// SIMATIC S7-200 project (STEP 7-Micro/WIN), CPU 226 CN REL 02.01

SYMBOL_TABLE 用户定义1
T_177            T177     // M25.1动作计时(2)
T_59             T59      // Y轴原点行程开关动作计时
T_83             T83      // M25.1动作计时(1)
T_71             T71      // M28.1动作计时(3)
T_70             T70      // M28.1动作计时(2)
T_69             T69      // M28.1动作计时(1)
T_185            T185     // PH1动作计时
T_180            T180     // PH2不动作计时
T_190            T190     // SL5动作延时
T_81             T81      // M26.0动作计时
T_82             T82      // 夹紧装置电磁阀松开线圈动作计时
SA2              I0.0     // 1=板链线与机械手联锁,0=板链线单独
SF3              I0.1     // 板链线/机械手联锁启动
SS3              I0.2     // 板链线/机械手联锁停止
SB_1             I0.3     // 板链线反转点动
SB_2             I0.4     // X轴Y轴伺服回原点
SB_3             I0.5     // 故障解除
KA1              I0.6     // 板链线变频故障
PH1              I0.7     // 板链线产品到位
PH2              I1.0     // 差速链工装板有无产品
SL1              I1.1     // X轴伺服左极限
SL2              I1.2     // X轴伺服原点(常闭触点输入)
SL3              I1.3     // X轴伺服右极限
SL4              I1.4     // Y轴伺服上极限
SL5              I1.5     // Y轴伺服原点(常闭触点输入)
SL6              I1.6     // Y轴伺服下极限
SL7              I1.7     // 板链线夹具到位
SL8              I2.0     // 板链线下线保护
SL11             I2.1     // 差速链线工装板后边沿
SL12             I2.2     // 差速链线工装板前边沿
SP1              I2.3     // Y轴提升气缸提升到位
SP2              I2.4     // Y轴提升气缸下降到位
SP3              I2.5     // Y轴旋转气缸旋转到位
SP4              I2.6     // Y轴旋转气缸复位到位
SP5              I2.7     // X轴旋转气缸旋转到位
ASD1_SRDY        I3.0     // X轴伺服准备完毕
ASD1_ZSPD        I3.1     // X轴伺服零速状态
ASD1_TPOS        I3.2     // X轴伺服位置软限位
ASD1_ALRM        I3.3     // X轴伺服报警
ASD2_SRDY        I3.4     // Y轴伺服准备完毕
ASD2_ZSPD        I3.5     // Y轴伺服零速状态
ASD2_TPOS        I3.6     // Y轴伺服位置软限位
ASD2_ALRM        I3.7     // Y轴伺服报警
SP6              I4.0     // X轴旋转气缸复位到位
SP7              I4.1     // 抓紧气缸抓紧(1)
SP8              I4.2     // 抓紧气缸抓紧(2)
SP9              I4.3     // 抓紧气缸抓紧(3)
SP10             I4.4     // 抓紧气缸抓紧(4)
SP11_14          I4.5     // 抓紧气缸松开
KP1              I4.6     // 压力过低报警
SJ1_7            I4.7     // 板链线/机械手急停
M0_0             M0.0     // 板链线/机械手联锁投入
M0_2             M0.2     // 板链线/机械手联锁运行上升延微分
M0_3             M0.3     // 板链线单独正转投入
M0_6             M0.6     // 故障蜂鸣告警
M0_7             M0.7     // 紧急停止蜂鸣告警
M1_0             M1.0     // 气压过低蜂鸣报警
M1_1             M1.1     // 蜂鸣报警消音
M1_2             M1.2     // 故障/气压过低蜂鸣报警汇总
M3_7             M3.7     // Y轴伺服在板链线/差速链线上空下移脉冲数逻辑运算错误
M4_0             M4.0     // 机械手Y轴伺服空闲位下降沿微分
M4_1             M4.1     // Y轴伺服在板链线上空下移动作保持
M5_1             M5.1     // Q0.0脉冲输出指令
M5_2             M5.2     // Q0.1脉冲输出指令
M7_1             M7.1     // M14.1下降沿微分
M7_2             M7.2     // 机械手总复位结束信号
M9_1             M9.1     // Q0.0脉冲控制子程序PTO0_CTRL的I_STOP参数
M9_2             M9.2     // Q0.0脉冲控制子程序PTO0_CTRL的D_STOP参数
M10_0            M10.0    // Q0.0脉冲控制子程序PTO0_CTRL执行完成标志
M11_0            M11.0    // 机械手点动模式
M11_3            M11.3    // X轴伺服点动
M11_4            M11.4    // Y轴伺服点动
M12_0            M12.0    // XY轴伺服原点回归点动
M12_1            M12.1    // X轴伺服原点回归点动
M12_2            M12.2    // Y轴伺服原点回归点动
M12_3            M12.3    // XY轴伺服原点回归停止
M12_4            M12.4    // X轴伺服原点回归保持
M12_5            M12.5    // Y轴伺服原点回归保持
M12_6            M12.6    // 机械手总复位
M12_7            M12.7    // 机械手总复位停止
M13_0            M13.0    // 机械手总复位进行中
M13_1            M13.1    // X轴伺服运行指示
M13_2            M13.2    // Y轴伺服运行指示
M14_0            M14.0    // Y轴提升气缸提升
M14_1            M14.1    // Y轴提升气缸下降
M14_2            M14.2    // Y轴旋转气缸旋转
M14_3            M14.3    // Y轴旋转气缸复位
M14_4            M14.4    // X轴旋转气缸旋转
M14_5            M14.5    // X轴旋转气缸复位
M14_6            M14.6    // 抓取气缸抓紧
M14_7            M14.7    // 抓取气缸松开
M15_0            M15.0    // X轴伺服回原点
M15_1            M15.1    // Y轴伺服回原点
M16_0            M16.0    // X轴从板链线上空移向差速链上空状态保持
M16_1            M16.1    // X轴走到一定位置时Y轴旋转没有到位则停止X轴移向差速链
M16_2            M16.2    // X轴走到一定位置时X轴旋转没有到位则停止X轴移向差速链
M16_3            M16.3    // X轴没有走到一定位置时不允许提升气缸下降
M17_0            M17.0    // 板链线/机械手联锁投入
M17_1            M17.1    // 联锁运行状态
M17_2            M17.2    // 板链线运行状态指示
M17_3            M17.3    // 设备故障指示
M17_4            M17.4    // 触摸屏紧急停止
M17_5            M17.5    // 控制柜硬急停/触摸屏软急停汇总
M17_6            M17.6    // 触摸屏上设备启动
M17_7            M17.7    // 触摸屏上设备停止
M18_0            M18.0    // 触摸屏上板链线反转点动
M18_1            M18.1    // 触摸屏上故障解除
M18_2            M18.2    // 触摸屏上报警消音
M18_3            M18.3    // 机械手X轴伺服空闲位(0=PTO忙,1=PTO空闲)
M18_4            M18.4    // 机械手Y轴伺服空闲位(0=PTO忙,1=PTO空闲)
M18_5            M18.5    // 触摸屏上机械手X轴伺服方向(0=移向差速链线,1=移向板链线)
M18_6            M18.6    // 触摸屏上机械手Y轴伺服方向(0=下移,1=上移)
M19_1            M19.1    // Q0.1脉冲控制子程序PTO1_CTRL的I_STOP参数
M19_2            M19.2    // Q0.1脉冲控制子程序PTO1_CTRL的D_STOP参数
M20_0            M20.0    // Q0.1脉冲控制子程序PTO1_CTRL执行完成标志
M21_0            M21.0    // 板链线夹具前边沿到位
M21_1            M21.1    // 机械手抓紧气缸抓紧
M21_2            M21.2    // 联锁运行时Y轴提升气缸提升保持
M22_1            M22.1    // 抓紧气缸抓紧磁性开关(1)已经动作
M22_2            M22.2    // 抓紧气缸抓紧磁性开关(2)已经动作
M22_3            M22.3    // 抓紧气缸抓紧磁性开关(3)已经动作
M22_4            M22.4    // 抓紧气缸抓紧磁性开关(4)已经动作
M22_5            M22.5    // 抓紧气缸4个抓紧检测磁性开关已经动作
M22_6            M22.6    // 抓紧气缸4个抓紧检测磁性开关已经动作上升延
M22_7            M22.7    // Y轴提升气缸缩回保持
M23_0            M23.0    // 板链线停车等待差速链空工装板到位
M23_1            M23.1    // X轴伺服右移/X轴旋转气缸旋转/Y轴旋转气缸旋转
M24_0            M24.0    // X轴伺服右移到位
M24_1            M24.1    // Y轴伺服电机下移(3种产品3种位置,大约20mm左右)
M24_2            M24.2    // Y轴伺服在差速链上空从当前位置移至对应产品处
M24_3            M24.3    // Y轴伺服空闲上升延微分
M24_7            M24.7    // 点动模式上升沿微分
M25_0            M25.0    // Y轴伺服下移到位
M25_1            M25.1    // 夹紧装置电磁阀松开线圈动作保持
M26_0            M26.0    // Y轴伺服上移到原点
M26_1            M26.1    // 抓紧气缸松开上升延
M26_2            M26.2    // Y轴伺服下移方向信号
M27_0            M27.0    // Y轴伺服上移到位
M28_0            M28.0    // X轴伺服左移
M28_1            M28.1    // X轴原点回归信号保持
M28_3            M28.3    // Y轴原点回归信号保持
M29_0            M29.0    // Y轴伺服回原点后再下降到对应的Y轴高度
M30_0            M30.0    // 机械手处于初始状态
M31_0            M31.0    // 差速链阻挡器电磁阀下降线圈得电保持
M31_6            M31.6    // 手动停止PTO0脉冲输出标志
M31_7            M31.7    // 手动停止PTO0脉冲输出标志
ASD1_PLS         Q0.0     // X轴伺服位置脉冲
ASD2_PLS         Q0.1     // Y轴伺服位置脉冲
ASD1_SIGN        Q0.2     // X轴伺服方向(0=移向差速链线,1=移向板链线)
ASD2_SIGN        Q0.3     // Y轴伺服方向(0=下移,1=上移)
KA2              Q0.7     // 设备启动/故障蜂鸣告警
KA3              Q1.0     // 板链线运行状态
KA4              Q1.1     // 板链线变频器正转
KA5              Q1.2     // 板链线变频器反转
KA6              Q1.3     // 板链线/机械手联锁运行状态
KA7              Q1.4     // 机械手紧急停止
KA8              Q1.5     // Y轴提升气缸提升
KA9              Q1.6     // Y轴提升气缸下降
KA10             Q1.7     // 故障闪光告警
YV2_1            Q2.0     // Y轴旋转气缸旋转
YV2_2            Q2.1     // Y轴旋转气缸复位
YV3_1            Q2.2     // X轴旋转气缸旋转
YV3_2            Q2.3     // X轴旋转气缸复位
YV4_1            Q2.4     // 抓取气缸抓紧
YV4_2            Q2.5     // 抓取气缸松开
YV11             Q2.6     // 差速链线前阻挡器
YV12             Q2.7     // 差速链线后阻挡器
ASD1启动           Q3.0     // X轴伺服启动
ASD1脉冲清除         Q3.1     // X轴伺服脉冲清除
ASD1原点回归         Q3.2     // X轴伺服原点回归
ASD1故障复位         Q3.3     // X轴伺服故障复位
ASD2启动           Q3.4     // Y轴伺服启动
ASD2脉冲清除         Q3.5     // Y轴伺服脉冲清除
ASD2原点回归         Q3.6     // Y轴伺服原点回归
ASD2故障复位         Q3.7     // Y轴伺服故障复位
SM0_0            SM0.0    // 该位始终为1
SM0_1            SM0.1    // 第一个扫描周期为1
SM66_7           SM66.7   // PTO0空闲位：0=PTO忙，1=PTO空闲
SM67_7           SM67.7   // PTO0/PWM0有效位：1=有效
SM76_7           SM76.7   // PTO1空闲位：0=PTO忙，1=PTO空闲
SM77_7           SM77.7   // PTO1/PWM1有效位：1=有效
SMD_72           SMD72    // PTO0脉冲计数值
SMD_82           SMD82    // PTO1脉冲计数值
SMW_68           SMW68    // PTO0/PWM0周期
SMW_78           SMW78    // PTO1/PWM1周期
T_37             T37      // 板链线/机械手启动告警时间
T_38             T38      // 板链线单独正转启动告警时间
T_39             T39      // 故障蜂鸣报警之静音时间
T_40             T40      // 故障蜂鸣报警之鸣音时间
T_41             T41      // 急停蜂鸣报警之静音时间
T_42             T42      // 急停蜂鸣报警之鸣音时间
T_43             T43      // 气压过低蜂鸣报警之静音时间
T_44             T44      // 气压过低蜂鸣报警之鸣音时间
T_46             T46      // 下线保护光电开关动作计时
T_51             T51      // 夹紧电磁阀夹紧动作时间
T_54             T54      // X轴右移到位信号保持时间
T_55             T55      // 夹紧装置电磁阀松开线圈动作时间
T_57             T57      // X轴伺服左移延时
T_58             T58      // 原点行程开关动作时间
T_61             T61      // 差速链阻挡器电磁阀下降线圈得电时间
T_111            T111     // XY轴伺服加减速用的时钟脉冲
T_112            T112     // Y轴伺服点动计时
T_115            T115     // 触摸屏上板链线运行动画图片切换时间
T_131            T131     // YV4-1动作计时
T_132            T132     // Y轴提升气缸提升动作计时(1)
T_133            T133     // Y轴提升气缸提升动作计时(2)
T_134            T134     // YV3-1动作计时
T_135            T135     // M24.1动作计时
T_136            T136     // Y轴伺服上移计时
T_157            T157     // 机械手总复位时到达X轴Y轴原点计时
T_158            T158     // M4.1动作计时
T_175            T175     // 机械手到达Y轴原点计时
T_200            T200     // Y轴下移到位信号保持时间
T_210            T210     // 紧急停止复位后（就是解除了紧急停止）计时
T_247            T247     // 联锁运行计时
V308_1           V308.1   // Q0.0脉冲手动模式子程序PTO0_MAN的Run/Stop参数
V1308_1          V1308.1  // Q0.1脉冲手动模式子程序PTO1_MAN的Run/Stop参数
VB_1             VB1      // 变频器频率检测方式(VB1=0自动检测,VB1=1手动给定)
VB_300           VB300    // Q0.0脉冲控制子程序PTO0_CTRL的错误代码
VB_314           VB314    // Q0.0脉冲手动模式子程序PTO0_MAN的错误代码
VB_1300          VB1300   // Q0.1脉冲控制子程序PTO1_CTRL的错误代码
VB_1314          VB1314   // Q0.1脉冲手动模式子程序PTO1_MAN的错误代码
VD_108           VD108    // PLC自动检测到的变频器频率值
VD_150           VD150    // 手动给定的变频器的当前频率值
VD_154           VD154    // 变频器的有效当前频率值
VD_160           VD160    // 产品种类(1小号,2中号,3大号,4自定义)
VD_164           VD164    // 小号产品的中心高度
VD_168           VD168    // 小号产品的半径
VD_172           VD172    // 中号产品的中心高度
VD_176           VD176    // 中号产品的半径
VD_180           VD180    // 大号产品的中心高度
VD_184           VD184    // 大号产品的半径
VD_188           VD188    // 自定义产品的长度
VD_192           VD192    // 自定义产品的直径
VD_196           VD196    // 当前有效产品的长度
VD_200           VD200    // 当前有效产品的半径
VD_294           VD294    // PTO0脉冲计数值
VD_302           VD302    // Q0.0脉冲控制子程序PTO0_CTRL的C_Pos参数
VD_310           VD310    // Q0.0脉冲手动模式子程序PTO0_MAN的Speed参数
VD_316           VD316    // Q0.0脉冲手动模式子程序PTO0_MAN的C_Pos参数
VD_1294          VD1294   // PTO1脉冲计数值
VD_1302          VD1302   // Q0.1脉冲控制子程序PTO1_CTRL的C_Pos参数
VD_1310          VD1310   // Q0.1脉冲手动模式子程序PTO1_MAN的Speed参数
VD_1316          VD1316   // Q0.1脉冲手动模式子程序PTO1_MAN的C_Pos参数
VD_1900          VD1900   // 机械手X轴与板链线运行速度相等时X轴伺服脉冲与变频器频率的比值
VD_1904          VD1904   // 机械手X轴与板链线运行速度相等时X轴伺服脉冲的频率
VD_2000          VD2000   // 机械手X轴与板链线同步时的PTO0周期值(微秒，实数)
VD_2004          VD2004   // 机械手X轴与板链线同步时的PTO0周期计算中间值1
VD_2008          VD2008   // 机械手X轴与板链线同步时的PTO0周期计算中间值2
VD_2012          VD2012   // 机械手X轴与板链线同步时的PTO0周期值(微秒,双整数)
VD_3000          VD3000   // 机械手在X轴方向每行走1mm，需要给X轴伺服电机的脉冲数(实数)
VD_3004          VD3004   // 机械手X轴与板链线同步的行走需要的脉冲数(实数)
VD_3008          VD3008   // 机械手X轴与板链线同步的行走需要的脉冲数(双整数)
VD_3016          VD3016   // X轴伺服跟随板链线行走完成后到移动到位需要的脉冲数(实数)
VD_3020          VD3020   // X轴伺服跟随板链线行走完成后到移动到位需要的脉冲数(双整数)
VD_4000          VD4000   // 机械手在Y轴方向每行走1mm，需要给Y轴伺服电机的脉冲数
VD_5000          VD5000   // 小号产品对应的Y轴伺服电机脉冲数(实数)
VD_5004          VD5004   // 小号产品对应的Y轴伺服电机脉冲数(双整数)
VD_5008          VD5008   // 在差速链上空各种产品对应的机械手Y轴下移脉冲数
VD_5020          VD5020   // 中号产品对应的Y轴伺服电机脉冲数(实数)
VD_5024          VD5024   // 中号产品对应的Y轴伺服电机脉冲数(双整数)
VD_5040          VD5040   // 大号产品对应的Y轴伺服电机脉冲数(实数)
VD_5044          VD5044   // 大号产品对应的Y轴伺服电机脉冲数(双整数)
VD_5052          VD5052   // 在差速链线上空各种产品对应的机械手Y轴下移脉冲数(电子齿轮比分子为3)
VD_6004          VD6004   // 小号产品对应的在板链线上空的Y轴伺服脉冲数(实数)
VD_6008          VD6008   // 小号产品对应的在板链线上空的Y轴伺服脉冲数(双整数)
VD_6012          VD6012   // 在板链链线上空各种产品对应的机械手Y轴下移脉冲数(电子齿轮比分子为1)
VD_6016          VD6016   // 在板链链线上空各种产品对应的机械手Y轴下移脉冲数(电子齿轮比分子为3)
VD_6024          VD6024   // 中号产品对应的在板链线上空的Y轴伺服脉冲数(实数)
VD_6028          VD6028   // 中号产品对应的在板链线上空的Y轴伺服脉冲数(双整数)
VD_6044          VD6044   // 大号产品对应的在板链线上空的Y轴伺服脉冲数(实数)
VD_6048          VD6048   // 大号产品对应的在板链线上空的Y轴伺服脉冲数(双整数)
VW_290           VW290    // PTO0/PWM0周期
VW_1290          VW1290   // PTO1/PWM1周期
VW_2020          VW2020   // 机械手X轴与板链线同步时的PTO0周期值(微秒，整数)
VW_7080          VW7080   // 触摸屏上板链线运行动画状态存储器
VW_7090          VW7090   // 触摸屏上机械手运行动画状态存储器
END_SYMBOL_TABLE

ORGANIZATION_BLOCK 总体控制:OB1
TITLE=总体控制；
BEGIN
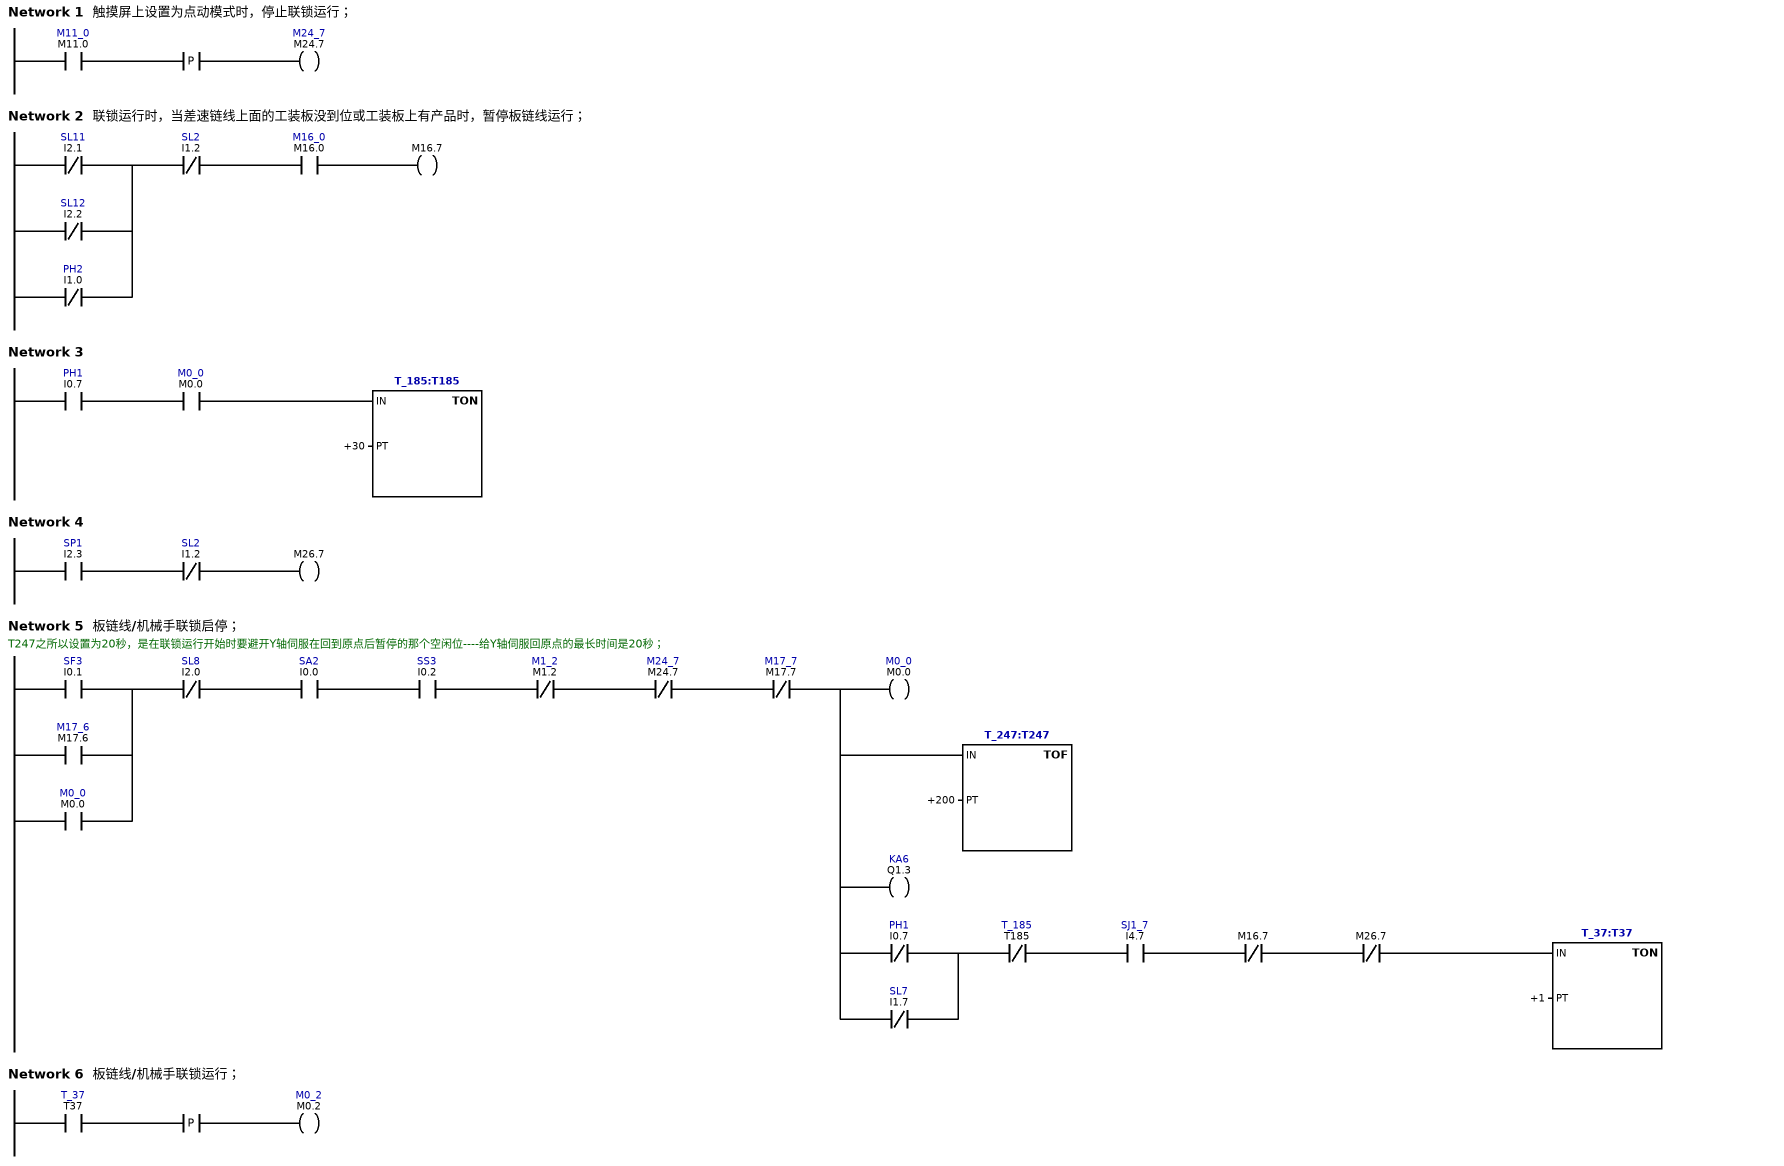
Network 1 // 触摸屏上设置为点动模式时，停止联锁运行；
LD     M11_0:M11.0
EU
=      M24_7:M24.7
Network 2 // 联锁运行时，当差速链线上面的工装板没到位或工装板上有产品时，暂停板链线运行；
LDN    SL11:I2.1
ON     SL12:I2.2
ON     PH2:I1.0
AN     SL2:I1.2
A      M16_0:M16.0
=      M16.7
Network 3
LD     PH1:I0.7
A      M0_0:M0.0
TON    T_185:T185, +30
Network 4
LD     SP1:I2.3
AN     SL2:I1.2
=      M26.7
Network 5 // 板链线/机械手联锁启停；
// T247之所以设置为20秒，是在联锁运行开始时要避开Y轴伺服在回到原点后暂停的那个空闲位----给Y轴伺服回原点的最长时间是20秒；
LD     SF3:I0.1
O      M17_6:M17.6
O      M0_0:M0.0
AN     SL8:I2.0
A      SA2:I0.0
A      SS3:I0.2
AN     M1_2:M1.2
AN     M24_7:M24.7
AN     M17_7:M17.7
=      M0_0:M0.0
TOF    T_247:T247, +200
=      KA6:Q1.3
LDN    PH1:I0.7
ON     SL7:I1.7
ALD
AN     T_185:T185
A      SJ1_7:I4.7
AN     M16.7
AN     M26.7
TON    T_37:T37, +1
Network 6 // 板链线/机械手联锁运行；
LD     T_37:T37
EU
=      M0_2:M0.2
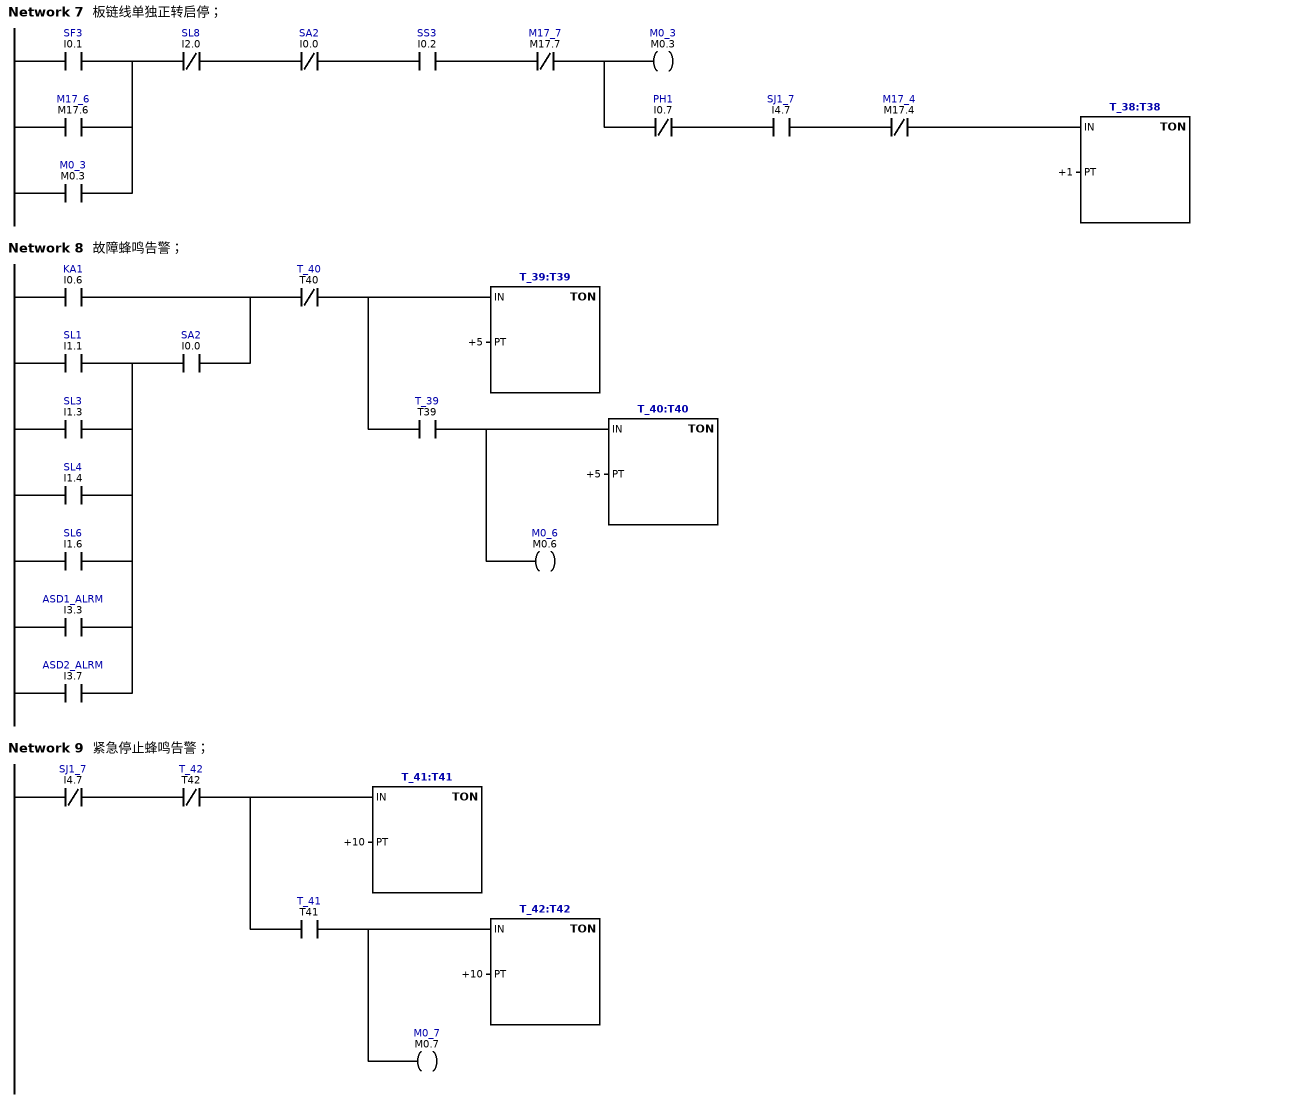
Network 7 // 板链线单独正转启停；
LD     SF3:I0.1
O      M17_6:M17.6
O      M0_3:M0.3
AN     SL8:I2.0
AN     SA2:I0.0
A      SS3:I0.2
AN     M17_7:M17.7
=      M0_3:M0.3
AN     PH1:I0.7
A      SJ1_7:I4.7
AN     M17_4:M17.4
TON    T_38:T38, +1
Network 8 // 故障蜂鸣告警；
LD     KA1:I0.6
LD     SL1:I1.1
O      SL3:I1.3
O      SL4:I1.4
O      SL6:I1.6
O      ASD1_ALRM:I3.3
O      ASD2_ALRM:I3.7
A      SA2:I0.0
OLD
AN     T_40:T40
TON    T_39:T39, +5
A      T_39:T39
TON    T_40:T40, +5
=      M0_6:M0.6
Network 9 // 紧急停止蜂鸣告警；
LDN    SJ1_7:I4.7
AN     T_42:T42
TON    T_41:T41, +10
A      T_41:T41
TON    T_42:T42, +10
=      M0_7:M0.7
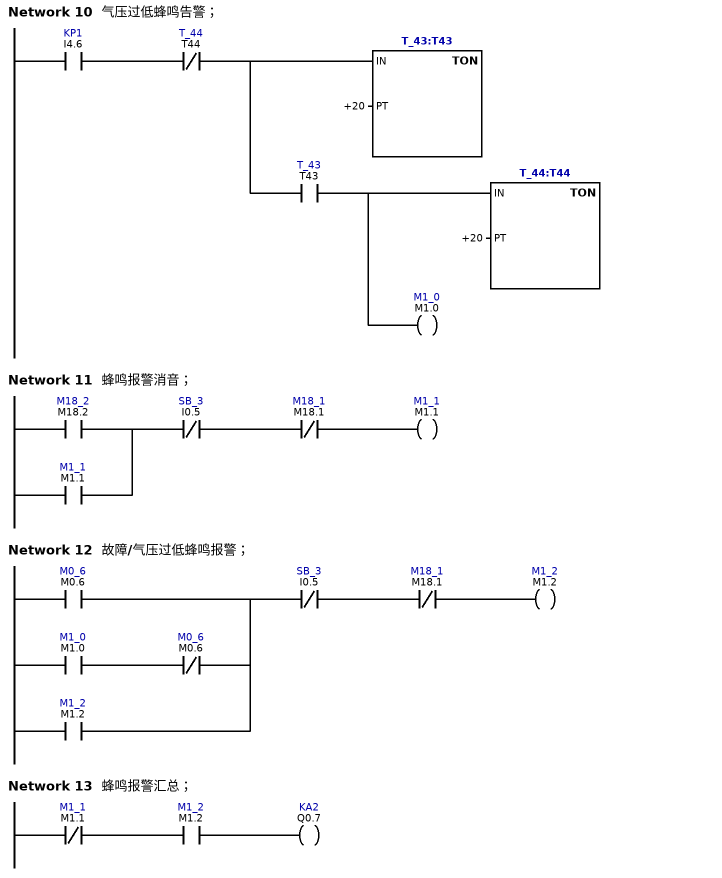
Network 10 // 气压过低蜂鸣告警；
LD     KP1:I4.6
AN     T_44:T44
TON    T_43:T43, +20
A      T_43:T43
TON    T_44:T44, +20
=      M1_0:M1.0
Network 11 // 蜂鸣报警消音；
LD     M18_2:M18.2
O      M1_1:M1.1
AN     SB_3:I0.5
AN     M18_1:M18.1
=      M1_1:M1.1
Network 12 // 故障/气压过低蜂鸣报警；
LD     M0_6:M0.6
LD     M1_0:M1.0
AN     M0_6:M0.6
OLD
O      M1_2:M1.2
AN     SB_3:I0.5
AN     M18_1:M18.1
=      M1_2:M1.2
Network 13 // 蜂鸣报警汇总；
LDN    M1_1:M1.1
A      M1_2:M1.2
=      KA2:Q0.7
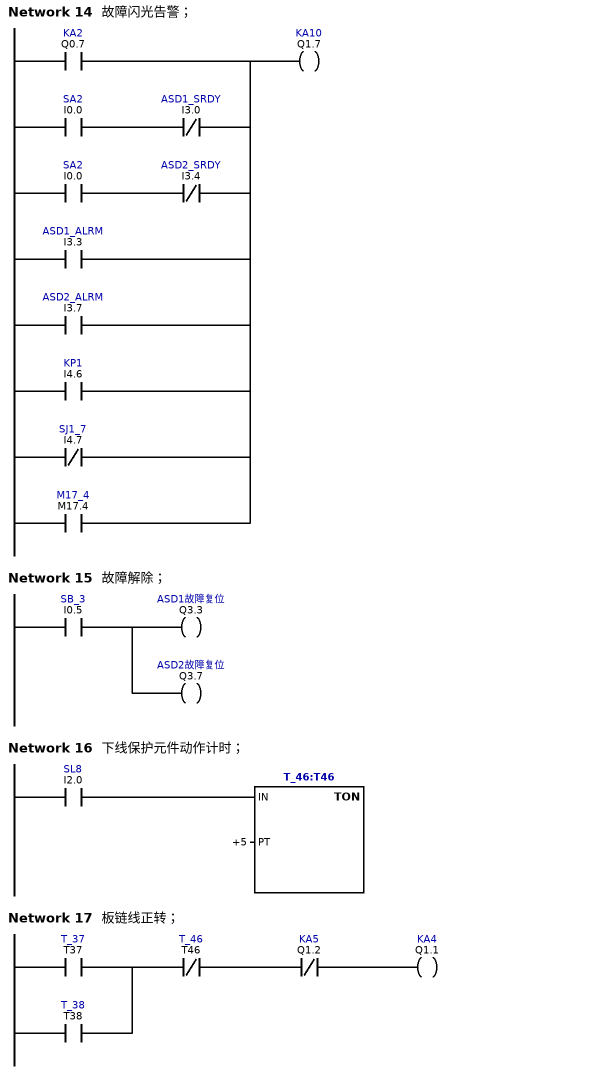
Network 14 // 故障闪光告警；
LD     KA2:Q0.7
LD     SA2:I0.0
AN     ASD1_SRDY:I3.0
OLD
LD     SA2:I0.0
AN     ASD2_SRDY:I3.4
OLD
O      ASD1_ALRM:I3.3
O      ASD2_ALRM:I3.7
O      KP1:I4.6
ON     SJ1_7:I4.7
O      M17_4:M17.4
=      KA10:Q1.7
Network 15 // 故障解除；
LD     SB_3:I0.5
=      ASD1故障复位:Q3.3
=      ASD2故障复位:Q3.7
Network 16 // 下线保护元件动作计时；
LD     SL8:I2.0
TON    T_46:T46, +5
Network 17 // 板链线正转；
LD     T_37:T37
O      T_38:T38
AN     T_46:T46
AN     KA5:Q1.2
=      KA4:Q1.1
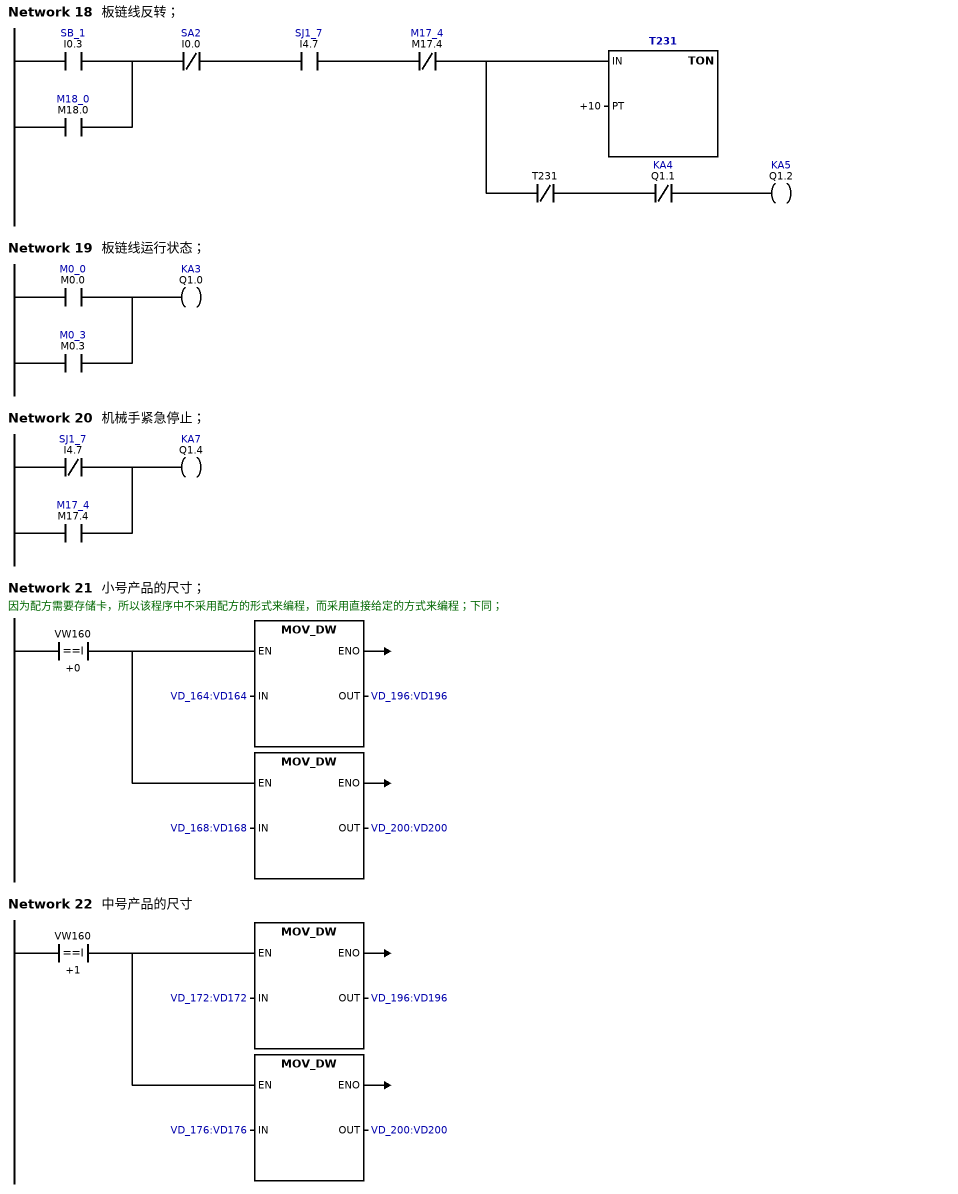
Network 18 // 板链线反转；
LD     SB_1:I0.3
O      M18_0:M18.0
AN     SA2:I0.0
A      SJ1_7:I4.7
AN     M17_4:M17.4
TON    T231, +10
AN     T231
AN     KA4:Q1.1
=      KA5:Q1.2
Network 19 // 板链线运行状态；
LD     M0_0:M0.0
O      M0_3:M0.3
=      KA3:Q1.0
Network 20 // 机械手紧急停止；
LDN    SJ1_7:I4.7
O      M17_4:M17.4
=      KA7:Q1.4
Network 21 // 小号产品的尺寸；
// 因为配方需要存储卡，所以该程序中不采用配方的形式来编程，而采用直接给定的方式来编程；下同；
LDW=   VW160, +0
MOVD   VD_164:VD164, VD_196:VD196
MOVD   VD_168:VD168, VD_200:VD200
Network 22 // 中号产品的尺寸
LDW=   VW160, +1
MOVD   VD_172:VD172, VD_196:VD196
MOVD   VD_176:VD176, VD_200:VD200
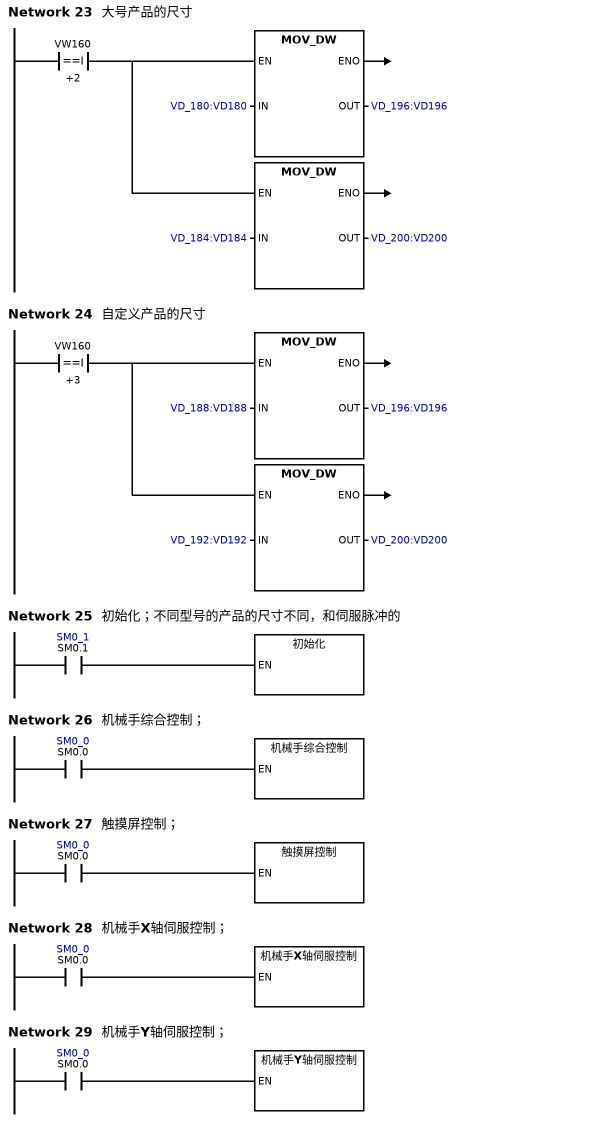
Network 23 // 大号产品的尺寸
LDW=   VW160, +2
MOVD   VD_180:VD180, VD_196:VD196
MOVD   VD_184:VD184, VD_200:VD200
Network 24 // 自定义产品的尺寸
LDW=   VW160, +3
MOVD   VD_188:VD188, VD_196:VD196
MOVD   VD_192:VD192, VD_200:VD200
Network 25 // 初始化；不同型号的产品的尺寸不同，和伺服脉冲的
LD     SM0_1:SM0.1
CALL   初始化:SBR0
Network 26 // 机械手综合控制；
LD     SM0_0:SM0.0
CALL   机械手综合控制:SBR2
Network 27 // 触摸屏控制；
LD     SM0_0:SM0.0
CALL   触摸屏控制:SBR3
Network 28 // 机械手X轴伺服控制；
LD     SM0_0:SM0.0
CALL   机械手X轴伺服控制:SBR11
Network 29 // 机械手Y轴伺服控制；
LD     SM0_0:SM0.0
CALL   机械手Y轴伺服控制:SBR12
END_ORGANIZATION_BLOCK

SUBROUTINE_BLOCK 初始化:SBR0
TITLE=初始化子程序；
// 设置一些中间变量，方便调试------重新下载程序后，这些变量仍然被正常赋值，不会变成零，不用重新赋值，节省调试时间；
BEGIN
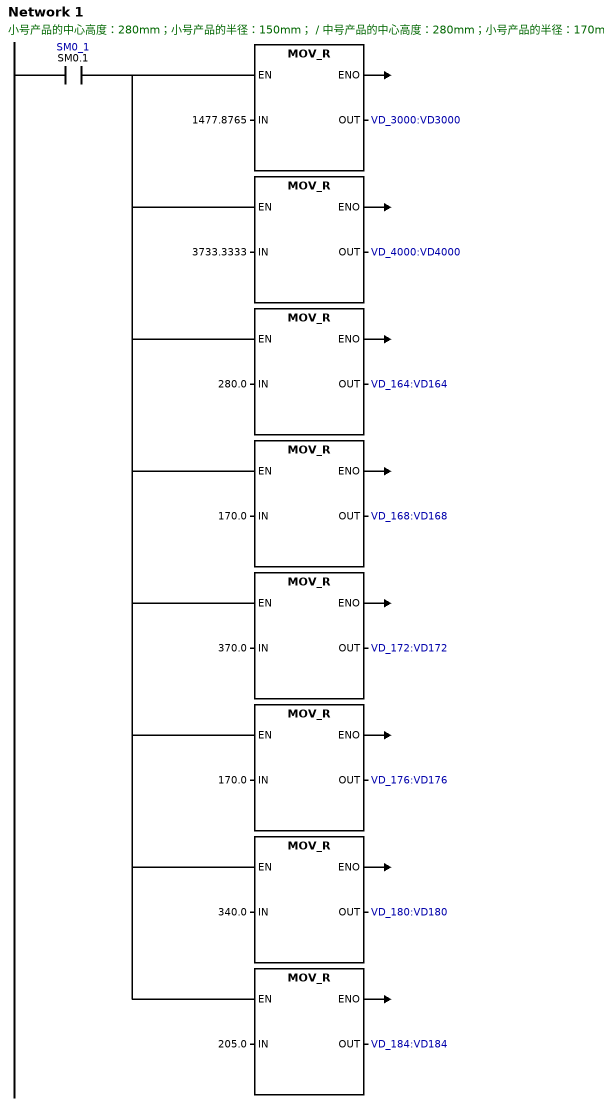
Network 1
// 小号产品的中心高度：280mm；小号产品的半径：150mm；
// 中号产品的中心高度：280mm；小号产品的半径：170mm；
// 大号产品的中心高度：340mm；小号产品的半径：205mm；
LD     SM0_1:SM0.1
MOVR   1477.8765, VD_3000:VD3000
MOVR   3733.3333, VD_4000:VD4000
MOVR   280.0, VD_164:VD164
MOVR   170.0, VD_168:VD168
MOVR   370.0, VD_172:VD172
MOVR   170.0, VD_176:VD176
MOVR   340.0, VD_180:VD180
MOVR   205.0, VD_184:VD184
END_SUBROUTINE_BLOCK

SUBROUTINE_BLOCK 机械手综合控制:SBR2
TITLE=机械手综合控制；
BEGIN
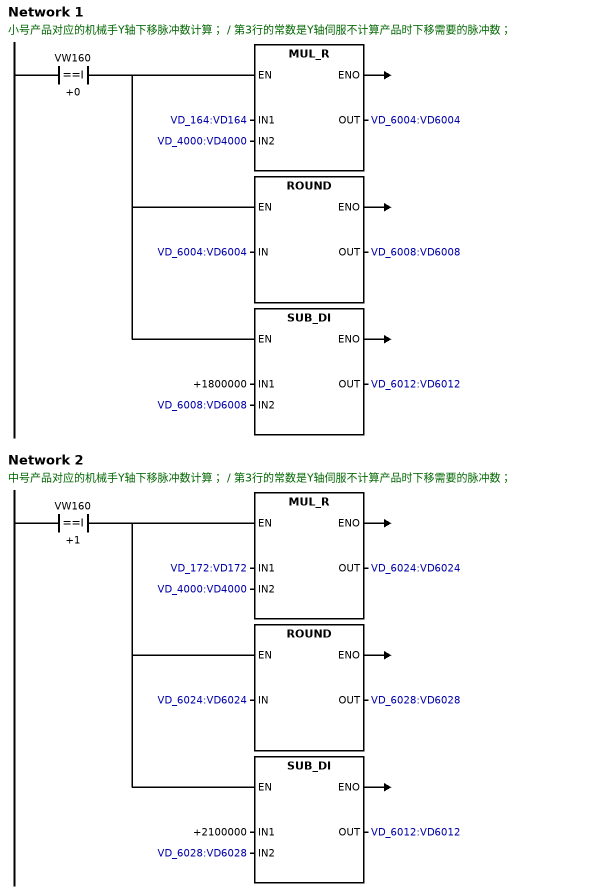
Network 1
// 小号产品对应的机械手Y轴下移脉冲数计算；
// 第3行的常数是Y轴伺服不计算产品时下移需要的脉冲数；
LDW=   VW160, +0
MOVR   VD_164:VD164, VD_6004:VD6004
*R     VD_4000:VD4000, VD_6004:VD6004
ROUND  VD_6004:VD6004, VD_6008:VD6008
MOVD   +1800000, VD_6012:VD6012
-D     VD_6008:VD6008, VD_6012:VD6012
Network 2
// 中号产品对应的机械手Y轴下移脉冲数计算；
// 第3行的常数是Y轴伺服不计算产品时下移需要的脉冲数；
LDW=   VW160, +1
MOVR   VD_172:VD172, VD_6024:VD6024
*R     VD_4000:VD4000, VD_6024:VD6024
ROUND  VD_6024:VD6024, VD_6028:VD6028
MOVD   +2100000, VD_6012:VD6012
-D     VD_6028:VD6028, VD_6012:VD6012
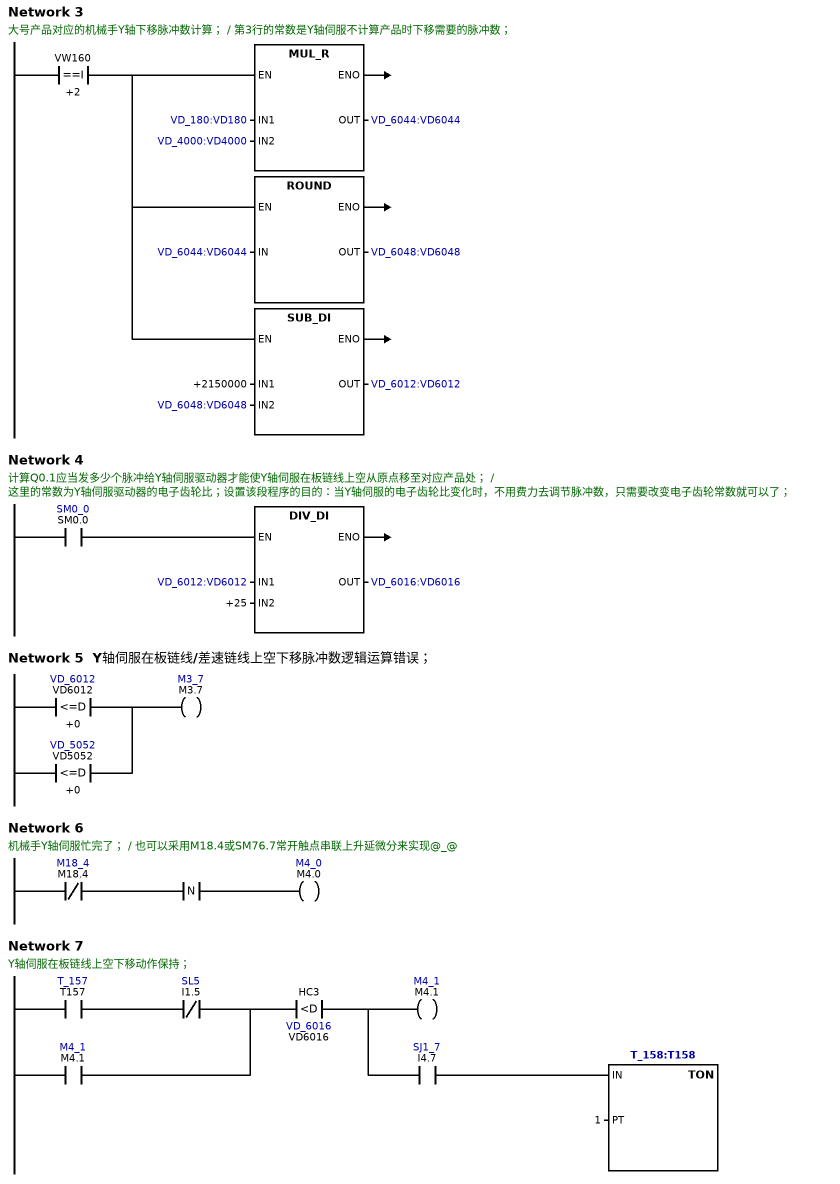
Network 3
// 大号产品对应的机械手Y轴下移脉冲数计算；
// 第3行的常数是Y轴伺服不计算产品时下移需要的脉冲数；
LDW=   VW160, +2
MOVR   VD_180:VD180, VD_6044:VD6044
*R     VD_4000:VD4000, VD_6044:VD6044
ROUND  VD_6044:VD6044, VD_6048:VD6048
MOVD   +2150000, VD_6012:VD6012
-D     VD_6048:VD6048, VD_6012:VD6012
Network 4
// 计算Q0.1应当发多少个脉冲给Y轴伺服驱动器才能使Y轴伺服在板链线上空从原点移至对应产品处；
// 这里的常数为Y轴伺服驱动器的电子齿轮比；设置该段程序的目的：当Y轴伺服的电子齿轮比变化时，不用费力去调节脉冲数，只需要改变电子齿轮常数就可以了；
LD     SM0_0:SM0.0
MOVD   VD_6012:VD6012, VD_6016:VD6016
/D     +25, VD_6016:VD6016
Network 5 // Y轴伺服在板链线/差速链线上空下移脉冲数逻辑运算错误；
LDD<=  VD_6012:VD6012, +0
OD<=   VD_5052:VD5052, +0
=      M3_7:M3.7
Network 6
// 机械手Y轴伺服忙完了；
// 也可以采用M18.4或SM76.7常开触点串联上升延微分来实现@_@
LDN    M18_4:M18.4
ED
=      M4_0:M4.0
Network 7
// Y轴伺服在板链线上空下移动作保持；
LD     T_157:T157
AN     SL5:I1.5
O      M4_1:M4.1
AD<    HC3, VD_6016:VD6016
=      M4_1:M4.1
A      SJ1_7:I4.7
TON    T_158:T158, 1
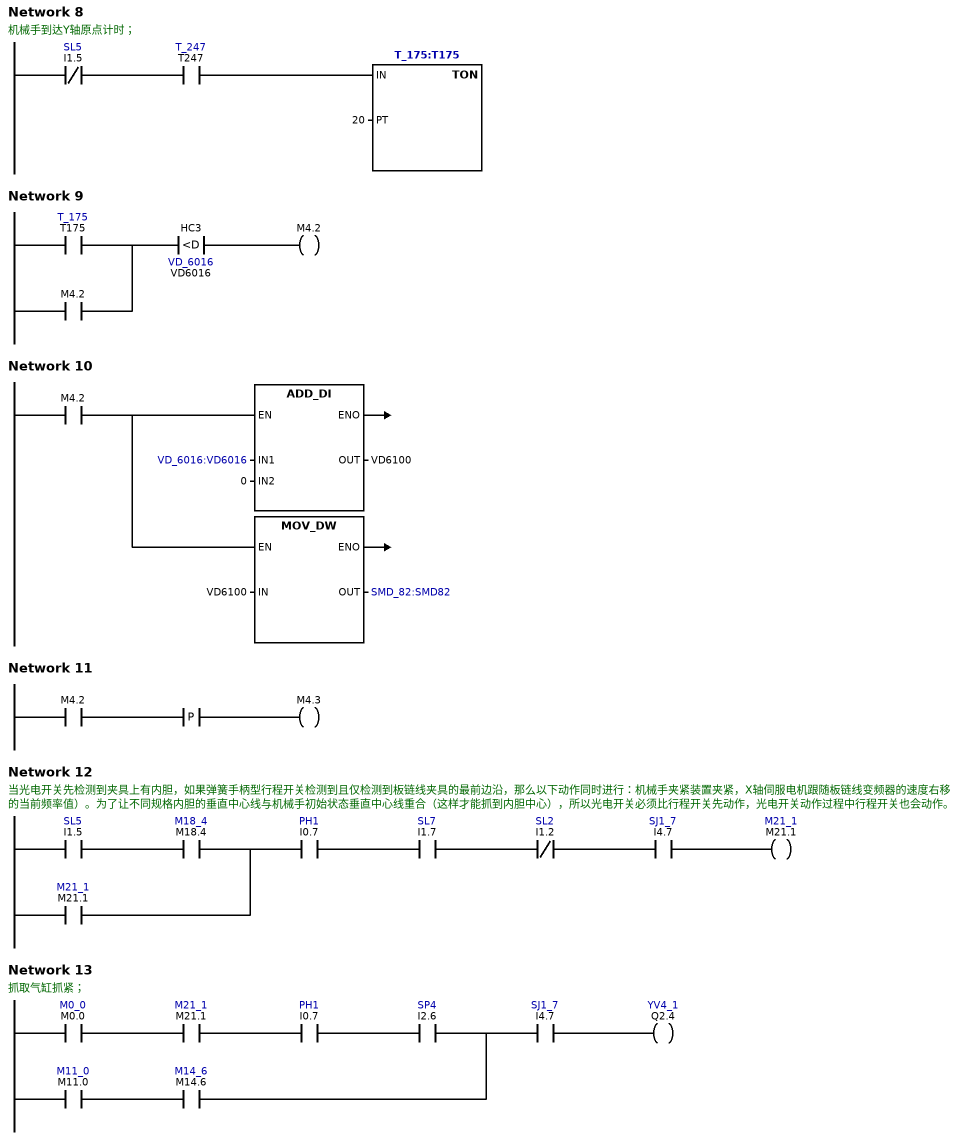
Network 8
// 机械手到达Y轴原点计时；
LDN    SL5:I1.5
A      T_247:T247
TON    T_175:T175, 20
Network 9
LD     T_175:T175
O      M4.2
AD<    HC3, VD_6016:VD6016
=      M4.2
Network 10
LD     M4.2
MOVD   VD_6016:VD6016, VD6100
+D     0, VD6100
MOVD   VD6100, SMD_82:SMD82
Network 11
LD     M4.2
EU
=      M4.3
Network 12
// 当光电开关先检测到夹具上有内胆，如果弹簧手柄型行程开关检测到且仅检测到板链线夹具的最前边沿，那么以下动作同时进行：机械手夹紧装置夹紧，X轴伺服电机跟随板链线变频器的速度右移（PLC与变频器通信得到变频器的当前频率值）。为了让不同规格内胆的垂直中心线与机械手初始状态垂直中心线重合（这样才能抓到内胆中心），所以光电开关必须比行程开关先动作，光电开关动作过程中行程开关也会动作。
LD     SL5:I1.5
A      M18_4:M18.4
O      M21_1:M21.1
A      PH1:I0.7
A      SL7:I1.7
AN     SL2:I1.2
A      SJ1_7:I4.7
=      M21_1:M21.1
Network 13
// 抓取气缸抓紧；
LD     M0_0:M0.0
A      M21_1:M21.1
A      PH1:I0.7
A      SP4:I2.6
LD     M11_0:M11.0
A      M14_6:M14.6
OLD
A      SJ1_7:I4.7
=      YV4_1:Q2.4
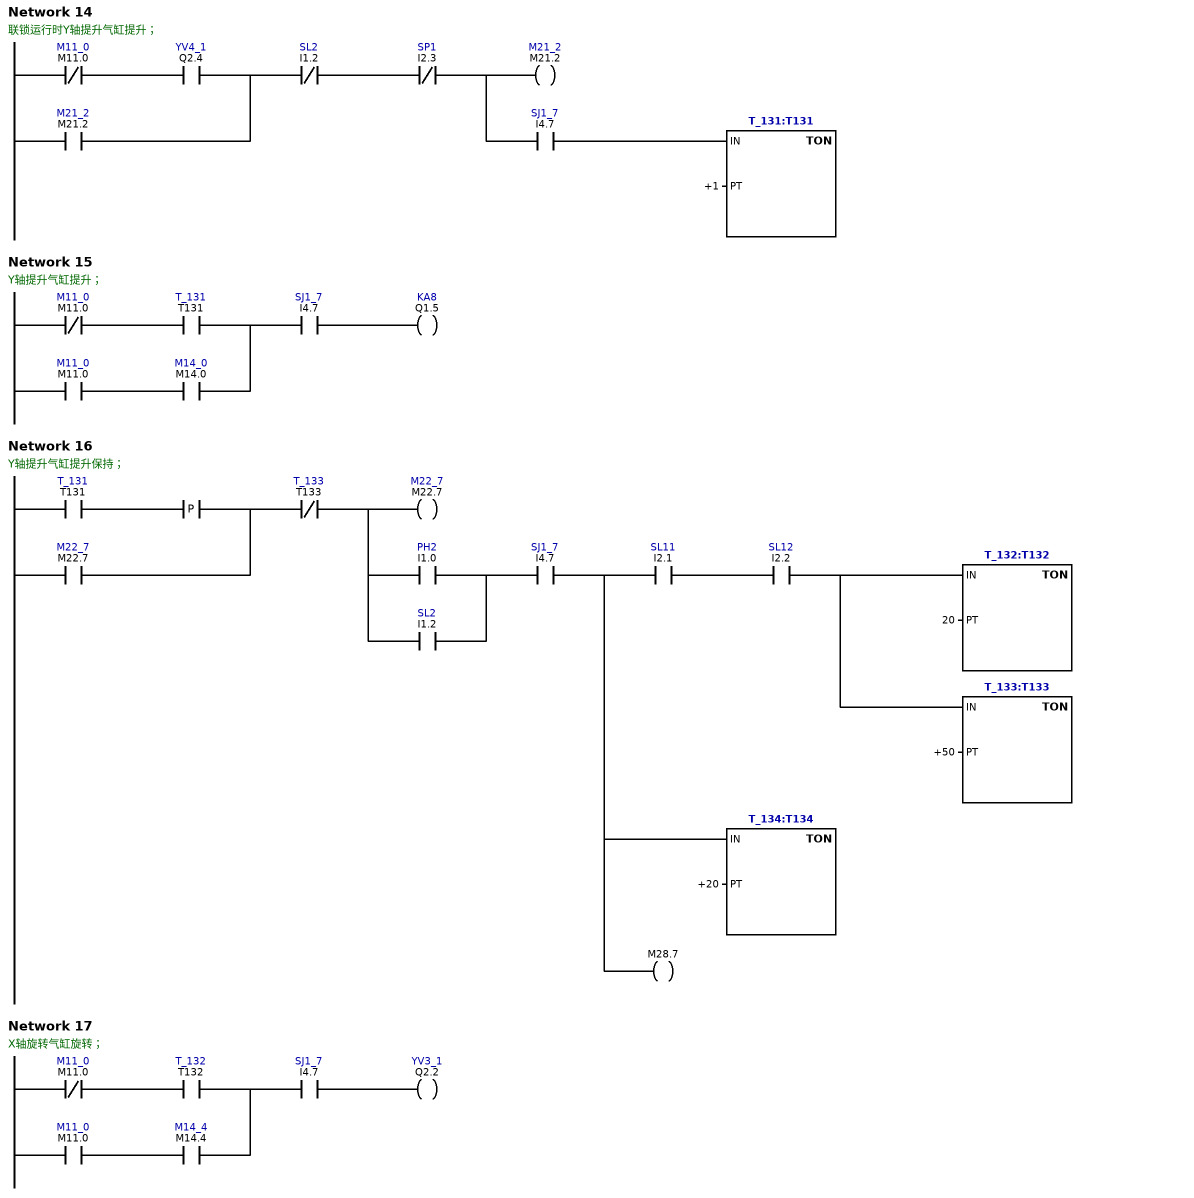
Network 14
// 联锁运行时Y轴提升气缸提升；
LDN    M11_0:M11.0
A      YV4_1:Q2.4
O      M21_2:M21.2
AN     SL2:I1.2
AN     SP1:I2.3
=      M21_2:M21.2
A      SJ1_7:I4.7
TON    T_131:T131, +1
Network 15
// Y轴提升气缸提升；
LDN    M11_0:M11.0
A      T_131:T131
LD     M11_0:M11.0
A      M14_0:M14.0
OLD
A      SJ1_7:I4.7
=      KA8:Q1.5
Network 16
// Y轴提升气缸提升保持；
LD     T_131:T131
EU
O      M22_7:M22.7
AN     T_133:T133
=      M22_7:M22.7
LD     PH2:I1.0
O      SL2:I1.2
A      SJ1_7:I4.7
ALD
LPS
A      SL11:I2.1
A      SL12:I2.2
TON    T_132:T132, 20
TON    T_133:T133, +50
LPP
TON    T_134:T134, +20
=      M28.7
Network 17
// X轴旋转气缸旋转；
LDN    M11_0:M11.0
A      T_132:T132
LD     M11_0:M11.0
A      M14_4:M14.4
OLD
A      SJ1_7:I4.7
=      YV3_1:Q2.2
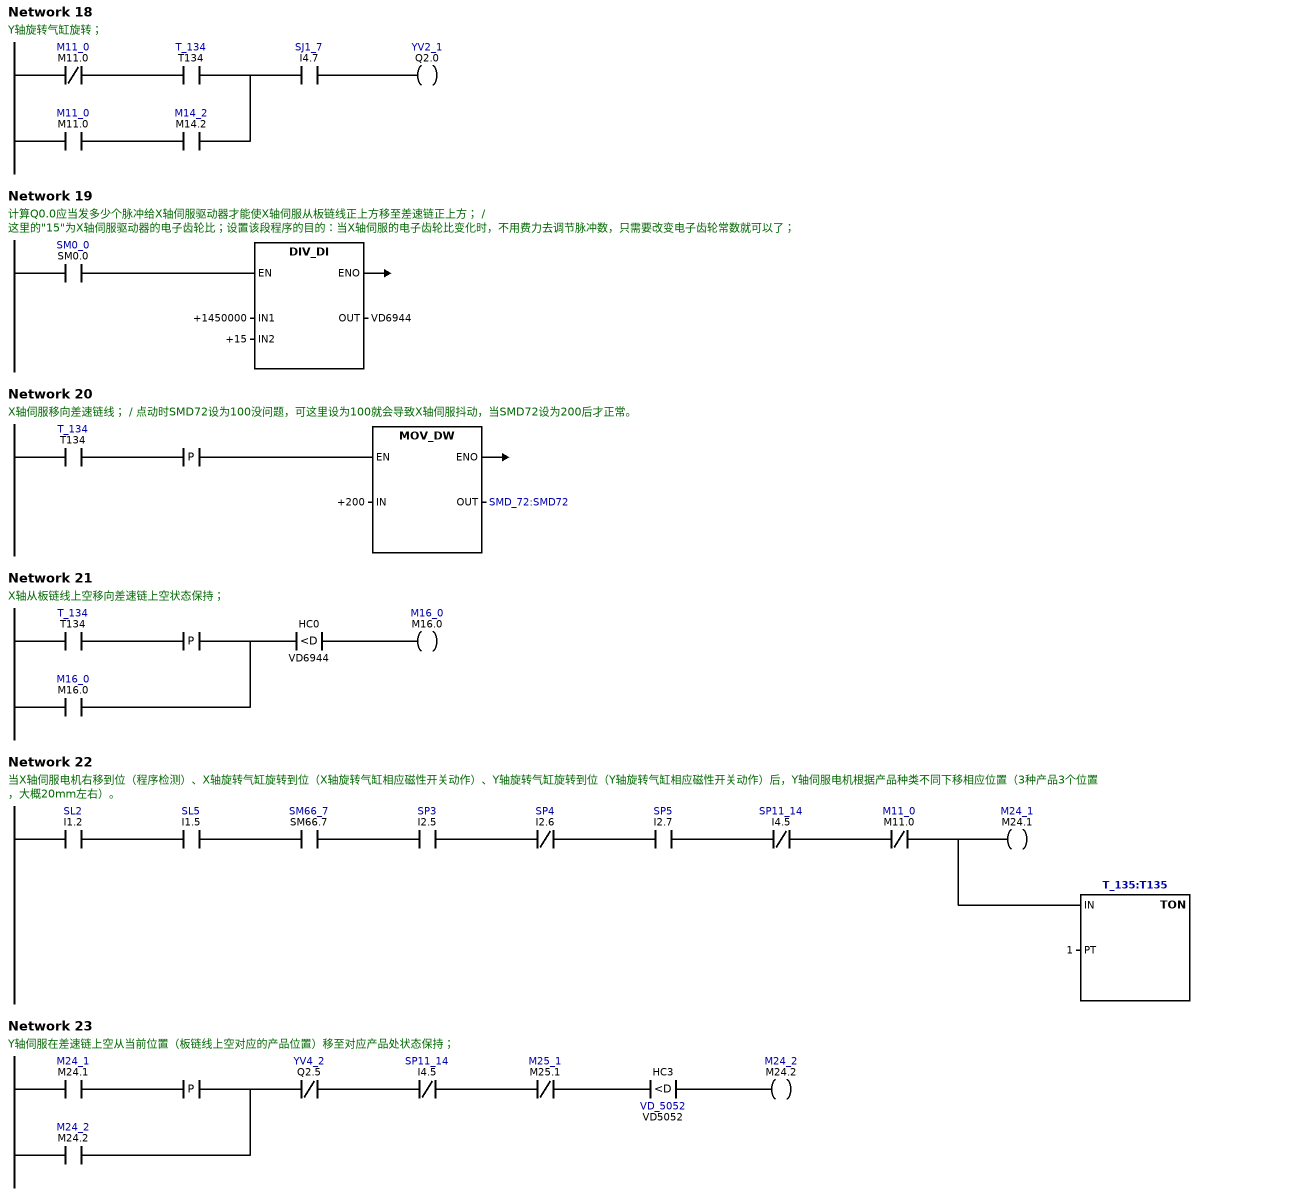
Network 18
// Y轴旋转气缸旋转；
LDN    M11_0:M11.0
A      T_134:T134
LD     M11_0:M11.0
A      M14_2:M14.2
OLD
A      SJ1_7:I4.7
=      YV2_1:Q2.0
Network 19
// 计算Q0.0应当发多少个脉冲给X轴伺服驱动器才能使X轴伺服从板链线正上方移至差速链正上方；
// 这里的"15"为X轴伺服驱动器的电子齿轮比；设置该段程序的目的：当X轴伺服的电子齿轮比变化时，不用费力去调节脉冲数，只需要改变电子齿轮常数就可以了；
LD     SM0_0:SM0.0
MOVD   +1450000, VD6944
/D     +15, VD6944
Network 20
// X轴伺服移向差速链线；
// 点动时SMD72设为100没问题，可这里设为100就会导致X轴伺服抖动，当SMD72设为200后才正常。
LD     T_134:T134
EU
MOVD   +200, SMD_72:SMD72
Network 21
// X轴从板链线上空移向差速链上空状态保持；
LD     T_134:T134
EU
O      M16_0:M16.0
AD<    HC0, VD6944
=      M16_0:M16.0
Network 22
// 当X轴伺服电机右移到位（程序检测）、X轴旋转气缸旋转到位（X轴旋转气缸相应磁性开关动作）、Y轴旋转气缸旋转到位（Y轴旋转气缸相应磁性开关动作）后，Y轴伺服电机根据产品种类不同下移相应位置（3种产品3个位置，大概20mm左右）。
LD     SL2:I1.2
A      SL5:I1.5
A      SM66_7:SM66.7
A      SP3:I2.5
AN     SP4:I2.6
A      SP5:I2.7
AN     SP11_14:I4.5
AN     M11_0:M11.0
=      M24_1:M24.1
TON    T_135:T135, 1
Network 23
// Y轴伺服在差速链上空从当前位置（板链线上空对应的产品位置）移至对应产品处状态保持；
LD     M24_1:M24.1
EU
O      M24_2:M24.2
AN     YV4_2:Q2.5
AN     SP11_14:I4.5
AN     M25_1:M25.1
AD<    HC3, VD_5052:VD5052
=      M24_2:M24.2
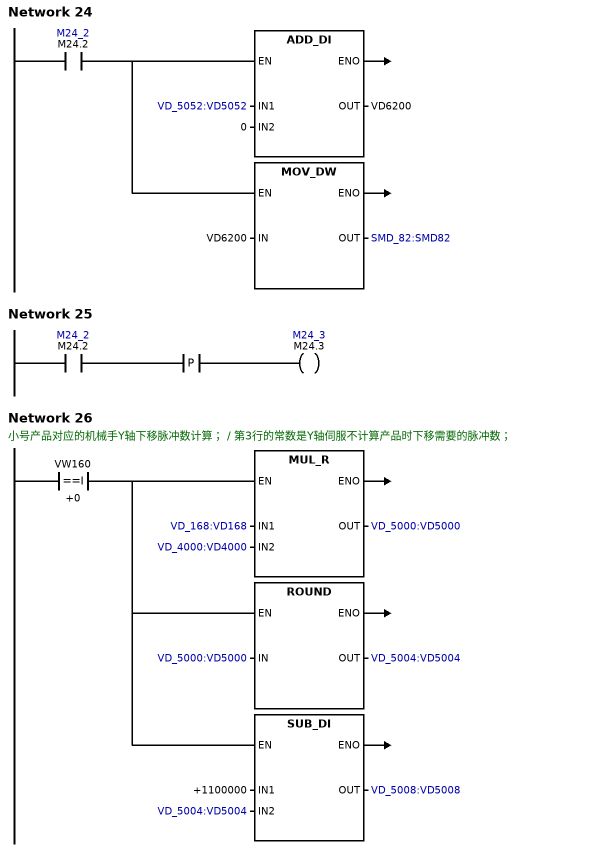
Network 24
LD     M24_2:M24.2
MOVD   VD_5052:VD5052, VD6200
+D     0, VD6200
MOVD   VD6200, SMD_82:SMD82
Network 25
LD     M24_2:M24.2
EU
=      M24_3:M24.3
Network 26
// 小号产品对应的机械手Y轴下移脉冲数计算；
// 第3行的常数是Y轴伺服不计算产品时下移需要的脉冲数；
LDW=   VW160, +0
MOVR   VD_168:VD168, VD_5000:VD5000
*R     VD_4000:VD4000, VD_5000:VD5000
ROUND  VD_5000:VD5000, VD_5004:VD5004
MOVD   +1100000, VD_5008:VD5008
-D     VD_5004:VD5004, VD_5008:VD5008
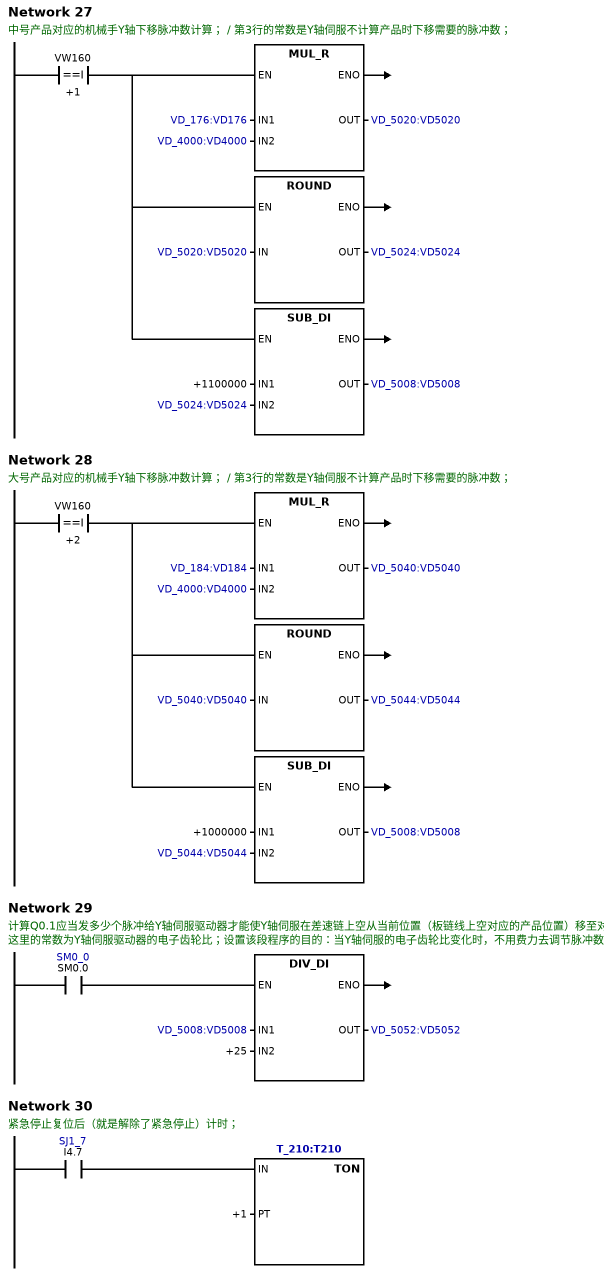
Network 27
// 中号产品对应的机械手Y轴下移脉冲数计算；
// 第3行的常数是Y轴伺服不计算产品时下移需要的脉冲数；
LDW=   VW160, +1
MOVR   VD_176:VD176, VD_5020:VD5020
*R     VD_4000:VD4000, VD_5020:VD5020
ROUND  VD_5020:VD5020, VD_5024:VD5024
MOVD   +1100000, VD_5008:VD5008
-D     VD_5024:VD5024, VD_5008:VD5008
Network 28
// 大号产品对应的机械手Y轴下移脉冲数计算；
// 第3行的常数是Y轴伺服不计算产品时下移需要的脉冲数；
LDW=   VW160, +2
MOVR   VD_184:VD184, VD_5040:VD5040
*R     VD_4000:VD4000, VD_5040:VD5040
ROUND  VD_5040:VD5040, VD_5044:VD5044
MOVD   +1000000, VD_5008:VD5008
-D     VD_5044:VD5044, VD_5008:VD5008
Network 29
// 计算Q0.1应当发多少个脉冲给Y轴伺服驱动器才能使Y轴伺服在差速链上空从当前位置（板链线上空对应的产品位置）移至对应产品处；
// 这里的常数为Y轴伺服驱动器的电子齿轮比；设置该段程序的目的：当Y轴伺服的电子齿轮比变化时，不用费力去调节脉冲数，只需要改变电子齿轮常数就可以了；
LD     SM0_0:SM0.0
MOVD   VD_5008:VD5008, VD_5052:VD5052
/D     +25, VD_5052:VD5052
Network 30
// 紧急停止复位后（就是解除了紧急停止）计时；
LD     SJ1_7:I4.7
TON    T_210:T210, +1
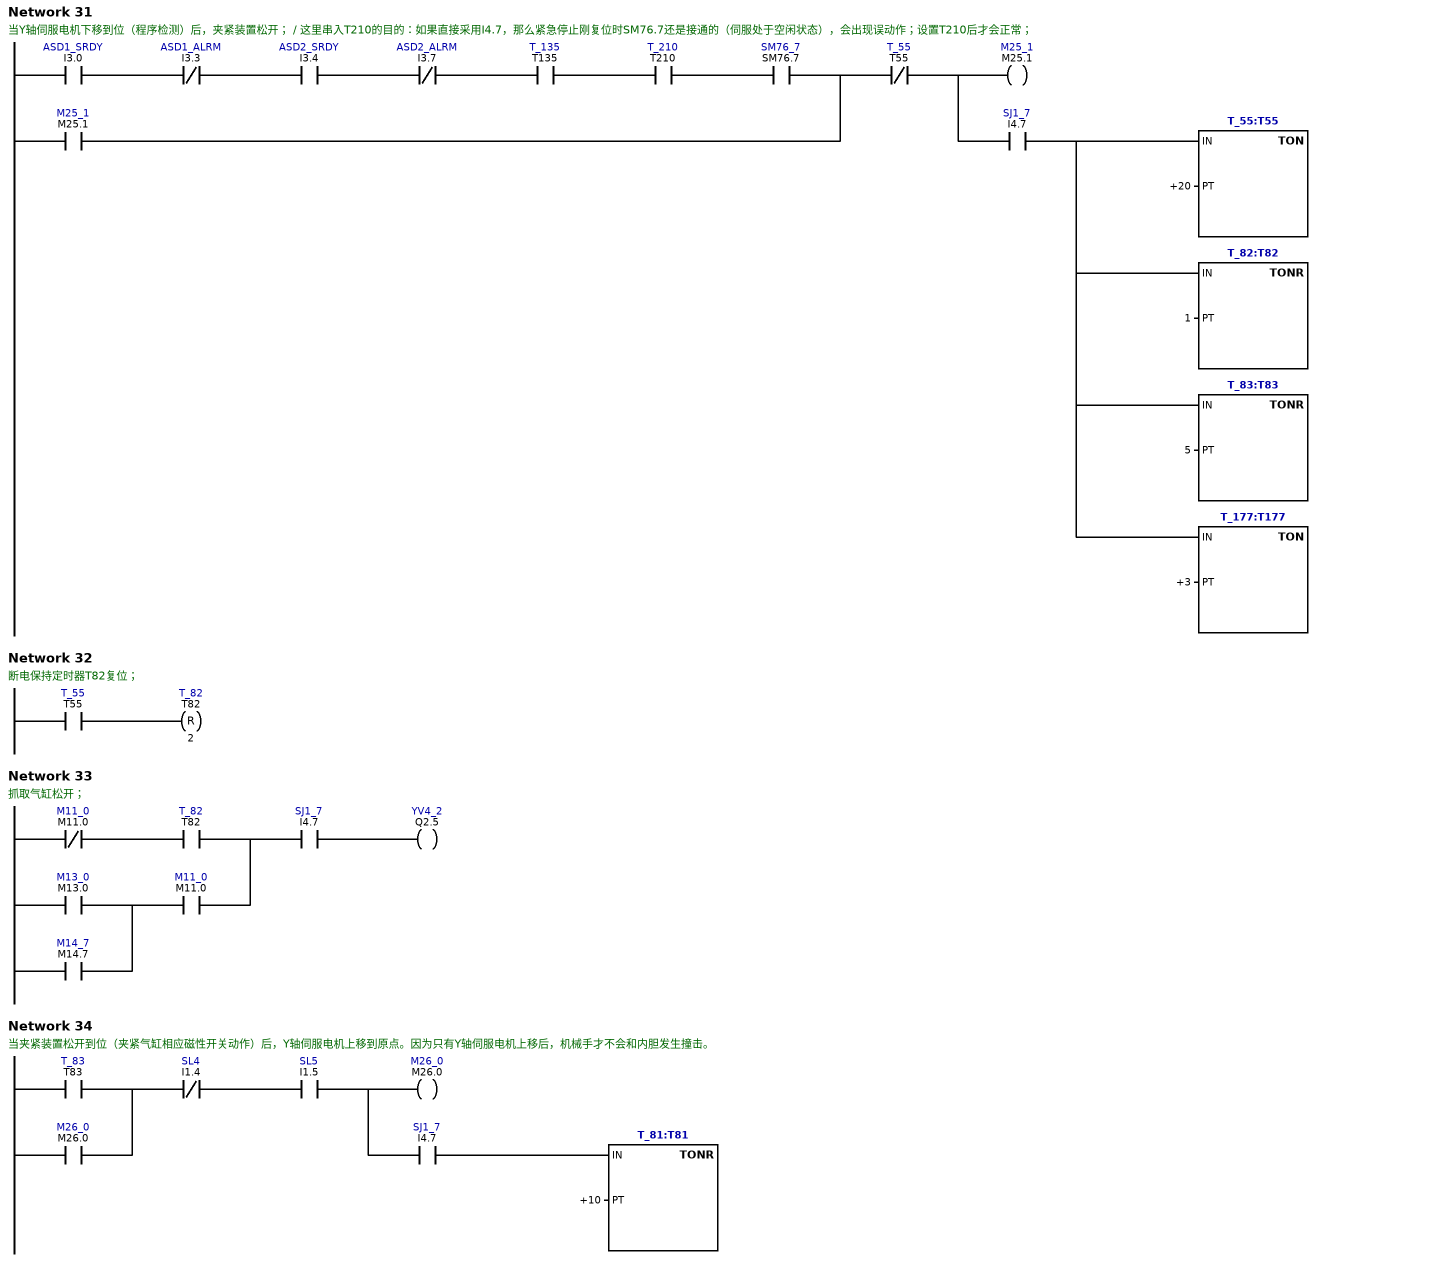
Network 31
// 当Y轴伺服电机下移到位（程序检测）后，夹紧装置松开；
// 这里串入T210的目的：如果直接采用I4.7，那么紧急停止刚复位时SM76.7还是接通的（伺服处于空闲状态），会出现误动作；设置T210后才会正常；
LD     ASD1_SRDY:I3.0
AN     ASD1_ALRM:I3.3
A      ASD2_SRDY:I3.4
AN     ASD2_ALRM:I3.7
A      T_135:T135
A      T_210:T210
A      SM76_7:SM76.7
O      M25_1:M25.1
AN     T_55:T55
=      M25_1:M25.1
A      SJ1_7:I4.7
TON    T_55:T55, +20
TONR   T_82:T82, 1
TONR   T_83:T83, 5
TON    T_177:T177, +3
Network 32
// 断电保持定时器T82复位；
LD     T_55:T55
R      T_82:T82, 2
Network 33
// 抓取气缸松开；
LDN    M11_0:M11.0
A      T_82:T82
LD     M13_0:M13.0
O      M14_7:M14.7
A      M11_0:M11.0
OLD
A      SJ1_7:I4.7
=      YV4_2:Q2.5
Network 34
// 当夹紧装置松开到位（夹紧气缸相应磁性开关动作）后，Y轴伺服电机上移到原点。因为只有Y轴伺服电机上移后，机械手才不会和内胆发生撞击。
LD     T_83:T83
O      M26_0:M26.0
AN     SL4:I1.4
A      SL5:I1.5
=      M26_0:M26.0
A      SJ1_7:I4.7
TONR   T_81:T81, +10
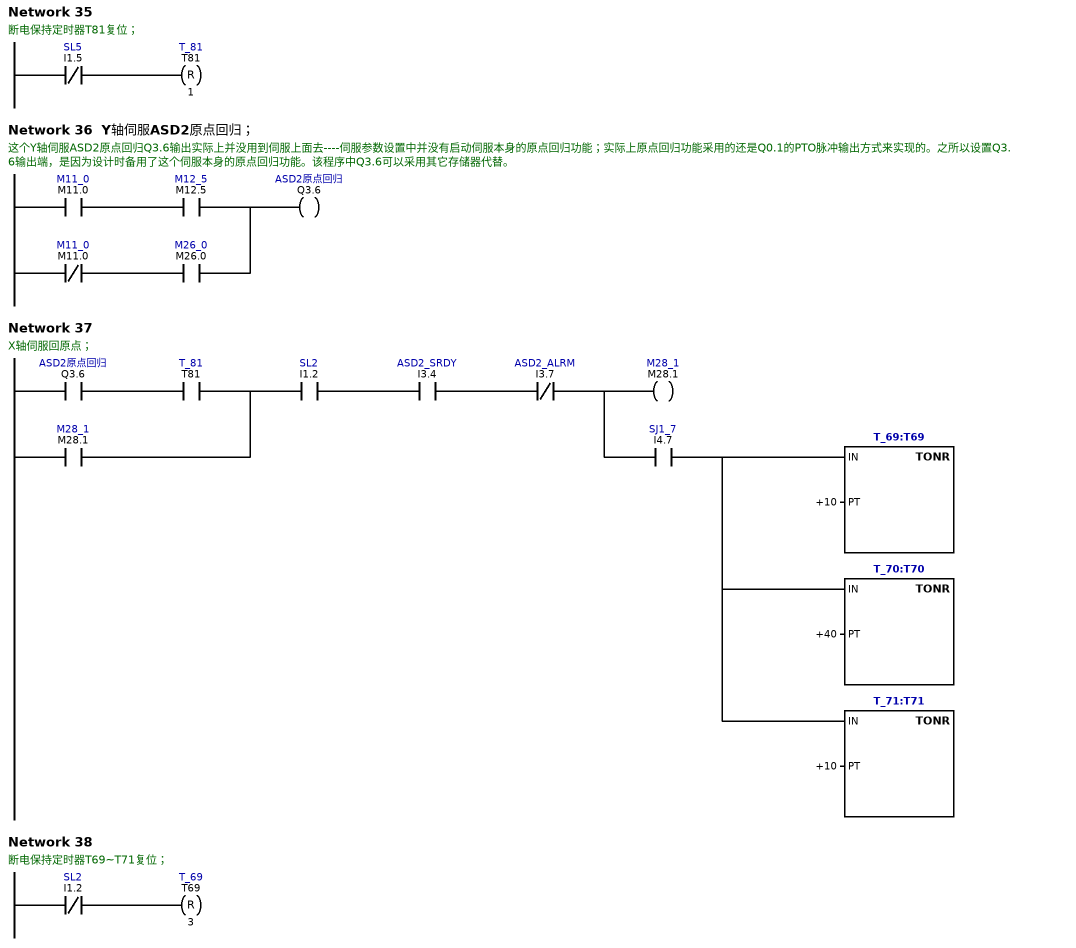
Network 35
// 断电保持定时器T81复位；
LDN    SL5:I1.5
R      T_81:T81, 1
Network 36 // Y轴伺服ASD2原点回归；
// 这个Y轴伺服ASD2原点回归Q3.6输出实际上并没用到伺服上面去----伺服参数设置中并没有启动伺服本身的原点回归功能；实际上原点回归功能采用的还是Q0.1的PTO脉冲输出方式来实现的。之所以设置Q3.6输出端，是因为设计时备用了这个伺服本身的原点回归功能。该程序中Q3.6可以采用其它存储器代替。
LD     M11_0:M11.0
A      M12_5:M12.5
LDN    M11_0:M11.0
A      M26_0:M26.0
OLD
=      ASD2原点回归:Q3.6
Network 37
// X轴伺服回原点；
LD     ASD2原点回归:Q3.6
A      T_81:T81
O      M28_1:M28.1
A      SL2:I1.2
A      ASD2_SRDY:I3.4
AN     ASD2_ALRM:I3.7
=      M28_1:M28.1
A      SJ1_7:I4.7
TONR   T_69:T69, +10
TONR   T_70:T70, +40
TONR   T_71:T71, +10
Network 38
// 断电保持定时器T69~T71复位；
LDN    SL2:I1.2
R      T_69:T69, 3
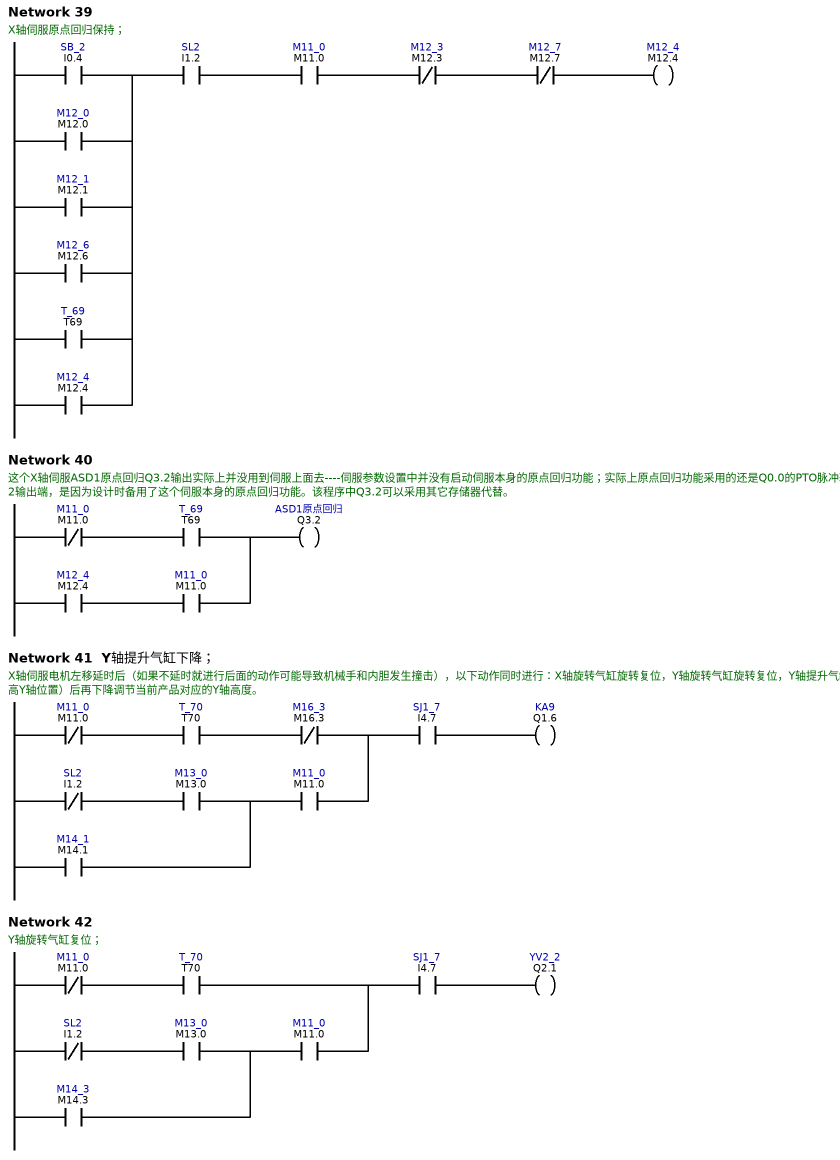
Network 39
// X轴伺服原点回归保持；
LD     SB_2:I0.4
O      M12_0:M12.0
O      M12_1:M12.1
O      M12_6:M12.6
O      T_69:T69
O      M12_4:M12.4
A      SL2:I1.2
A      M11_0:M11.0
AN     M12_3:M12.3
AN     M12_7:M12.7
=      M12_4:M12.4
Network 40
// 这个X轴伺服ASD1原点回归Q3.2输出实际上并没用到伺服上面去----伺服参数设置中并没有启动伺服本身的原点回归功能；实际上原点回归功能采用的还是Q0.0的PTO脉冲输出方式来实现的。之所以设置Q3.2输出端，是因为设计时备用了这个伺服本身的原点回归功能。该程序中Q3.2可以采用其它存储器代替。
LDN    M11_0:M11.0
A      T_69:T69
LD     M12_4:M12.4
A      M11_0:M11.0
OLD
=      ASD1原点回归:Q3.2
Network 41 // Y轴提升气缸下降；
// X轴伺服电机左移延时后（如果不延时就进行后面的动作可能导致机械手和内胆发生撞击），以下动作同时进行：X轴旋转气缸旋转复位，Y轴旋转气缸旋转复位，Y轴提升气缸伸出，Y轴伺服电机先回到Y轴原点（3种产品中的最高Y轴位置）后再下降调节当前产品对应的Y轴高度。
LDN    M11_0:M11.0
A      T_70:T70
AN     M16_3:M16.3
LDN    SL2:I1.2
A      M13_0:M13.0
O      M14_1:M14.1
A      M11_0:M11.0
OLD
A      SJ1_7:I4.7
=      KA9:Q1.6
Network 42
// Y轴旋转气缸复位；
LDN    M11_0:M11.0
A      T_70:T70
LDN    SL2:I1.2
A      M13_0:M13.0
O      M14_3:M14.3
A      M11_0:M11.0
OLD
A      SJ1_7:I4.7
=      YV2_2:Q2.1
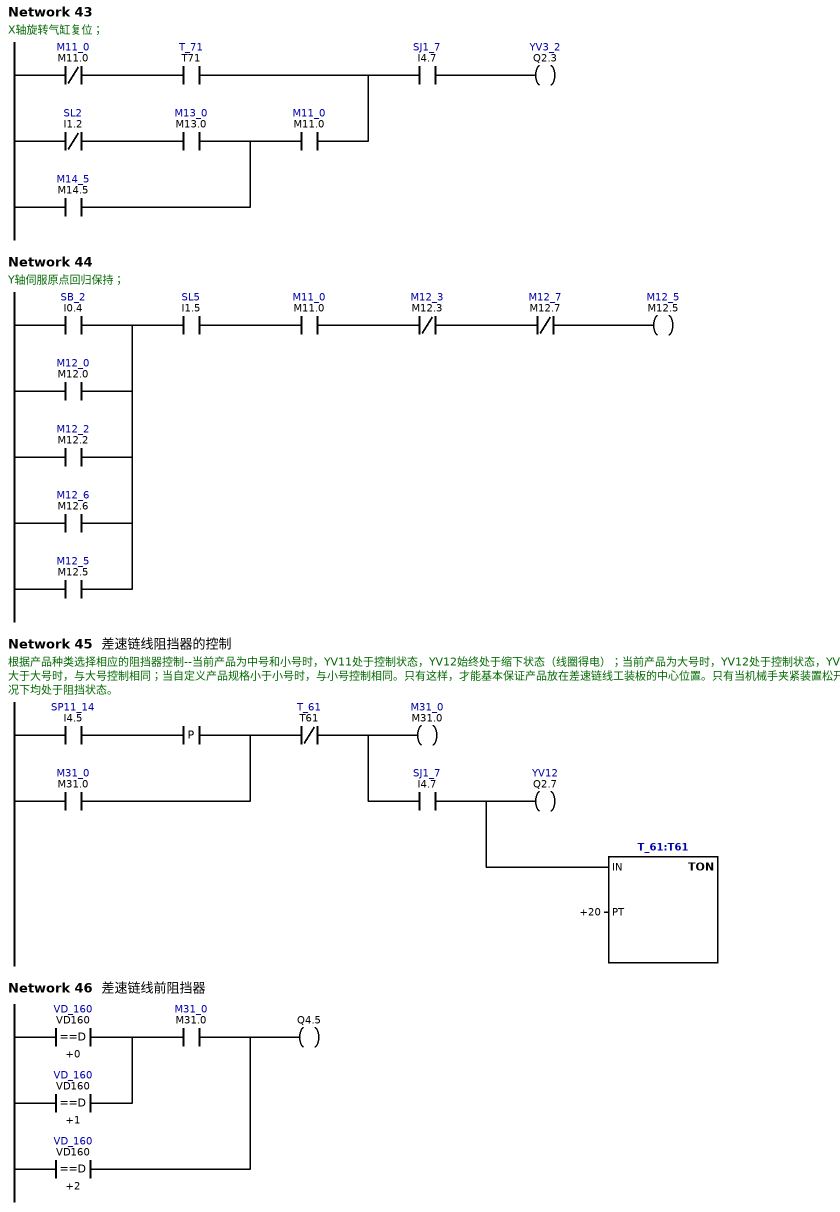
Network 43
// X轴旋转气缸复位；
LDN    M11_0:M11.0
A      T_71:T71
LDN    SL2:I1.2
A      M13_0:M13.0
O      M14_5:M14.5
A      M11_0:M11.0
OLD
A      SJ1_7:I4.7
=      YV3_2:Q2.3
Network 44
// Y轴伺服原点回归保持；
LD     SB_2:I0.4
O      M12_0:M12.0
O      M12_2:M12.2
O      M12_6:M12.6
O      M12_5:M12.5
A      SL5:I1.5
A      M11_0:M11.0
AN     M12_3:M12.3
AN     M12_7:M12.7
=      M12_5:M12.5
Network 45 // 差速链线阻挡器的控制
// 根据产品种类选择相应的阻挡器控制--当前产品为中号和小号时，YV11处于控制状态，YV12始终处于缩下状态（线圈得电）；当前产品为大号时，YV12处于控制状态，YV11始终处于缩下状态（线圈得电）；当自定义产品规格大于大号时，与大号控制相同；当自定义产品规格小于小号时，与小号控制相同。只有这样，才能基本保证产品放在差速链线工装板的中心位置。只有当机械手夹紧装置松开时，受控阻挡器才下降2秒左右处于放行状态，平常状况下均处于阻挡状态。
LD     SP11_14:I4.5
EU
O      M31_0:M31.0
AN     T_61:T61
=      M31_0:M31.0
A      SJ1_7:I4.7
=      YV12:Q2.7
TON    T_61:T61, +20
Network 46 // 差速链线前阻挡器
LDD=   VD_160:VD160, +0
OD=    VD_160:VD160, +1
A      M31_0:M31.0
OD=    VD_160:VD160, +2
=      Q4.5
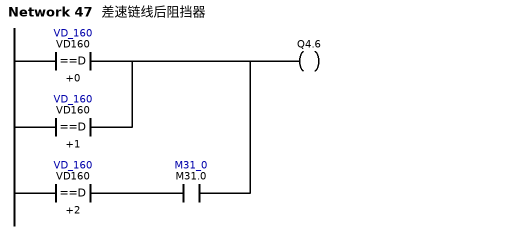
Network 47 // 差速链线后阻挡器
LDD=   VD_160:VD160, +0
OD=    VD_160:VD160, +1
LDD=   VD_160:VD160, +2
A      M31_0:M31.0
OLD
=      Q4.6
END_SUBROUTINE_BLOCK

SUBROUTINE_BLOCK 触摸屏控制:SBR3
TITLE=触摸屏控制；
// M17.6：触摸屏上设备启动；
// M17.7：触摸屏上设备停止；
// M18.0：触摸屏上板链线反转点动；
// M18.1：触摸屏上故障解除；
// M18.2：触摸屏上报警消音；
// M18.5：触摸屏上机械手X轴伺服电机转向(0=移向板链线,1=移向差速链线)
// M18.6：触摸屏上机械手Y轴伺服电机转向(0=下移,1=上移)
BEGIN
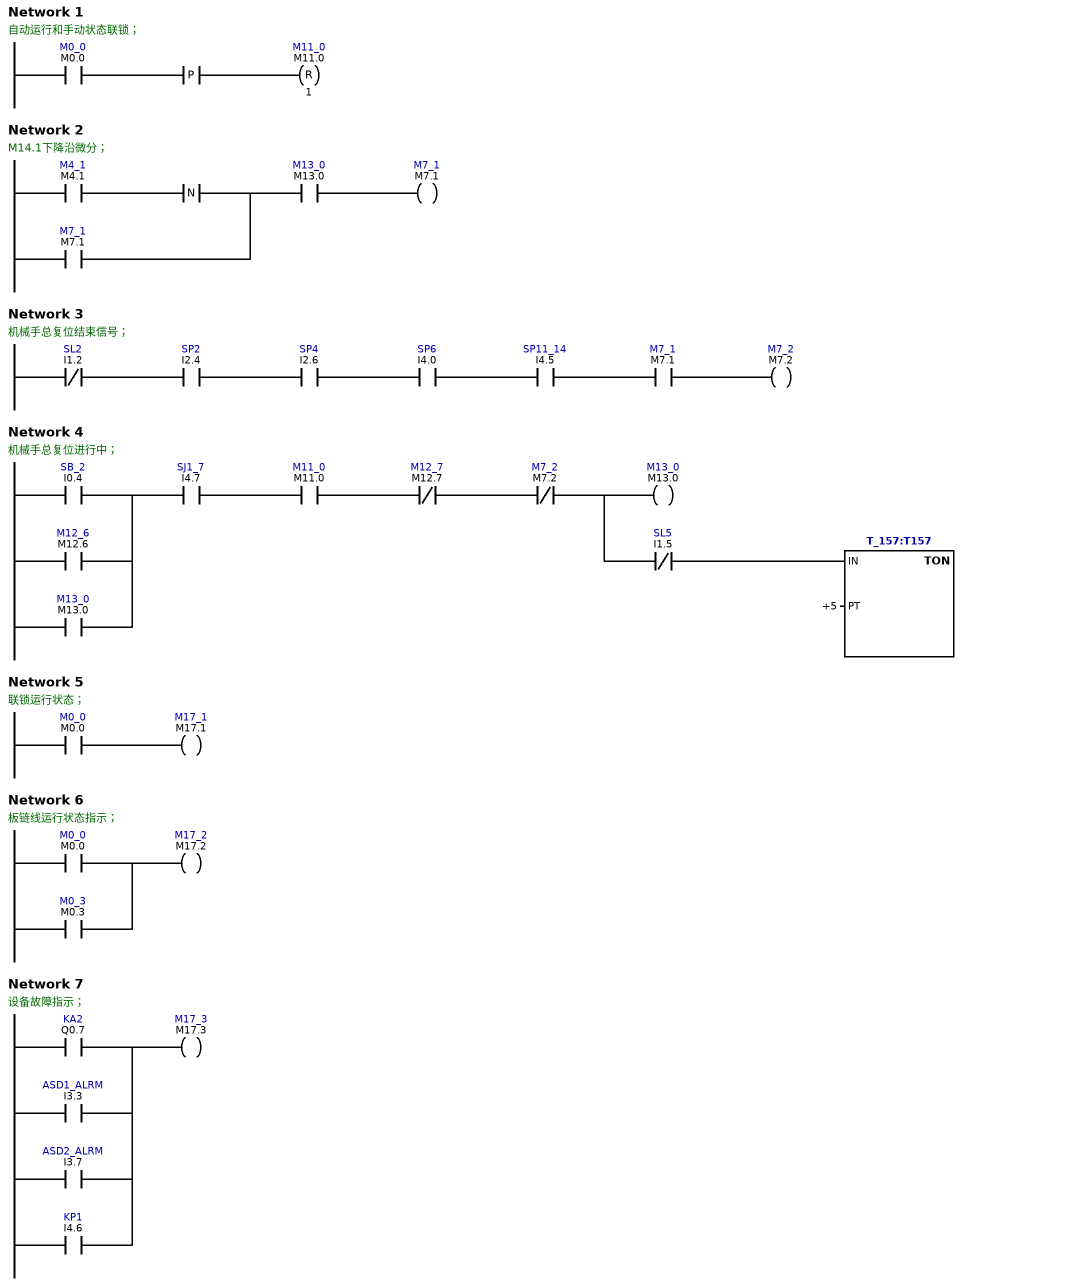
Network 1
// 自动运行和手动状态联锁；
LD     M0_0:M0.0
EU
R      M11_0:M11.0, 1
Network 2
// M14.1下降沿微分；
LD     M4_1:M4.1
ED
O      M7_1:M7.1
A      M13_0:M13.0
=      M7_1:M7.1
Network 3
// 机械手总复位结束信号；
LDN    SL2:I1.2
A      SP2:I2.4
A      SP4:I2.6
A      SP6:I4.0
A      SP11_14:I4.5
A      M7_1:M7.1
=      M7_2:M7.2
Network 4
// 机械手总复位进行中；
LD     SB_2:I0.4
O      M12_6:M12.6
O      M13_0:M13.0
A      SJ1_7:I4.7
A      M11_0:M11.0
AN     M12_7:M12.7
AN     M7_2:M7.2
=      M13_0:M13.0
AN     SL5:I1.5
TON    T_157:T157, +5
Network 5
// 联锁运行状态；
LD     M0_0:M0.0
=      M17_1:M17.1
Network 6
// 板链线运行状态指示；
LD     M0_0:M0.0
O      M0_3:M0.3
=      M17_2:M17.2
Network 7
// 设备故障指示；
LD     KA2:Q0.7
O      ASD1_ALRM:I3.3
O      ASD2_ALRM:I3.7
O      KP1:I4.6
=      M17_3:M17.3
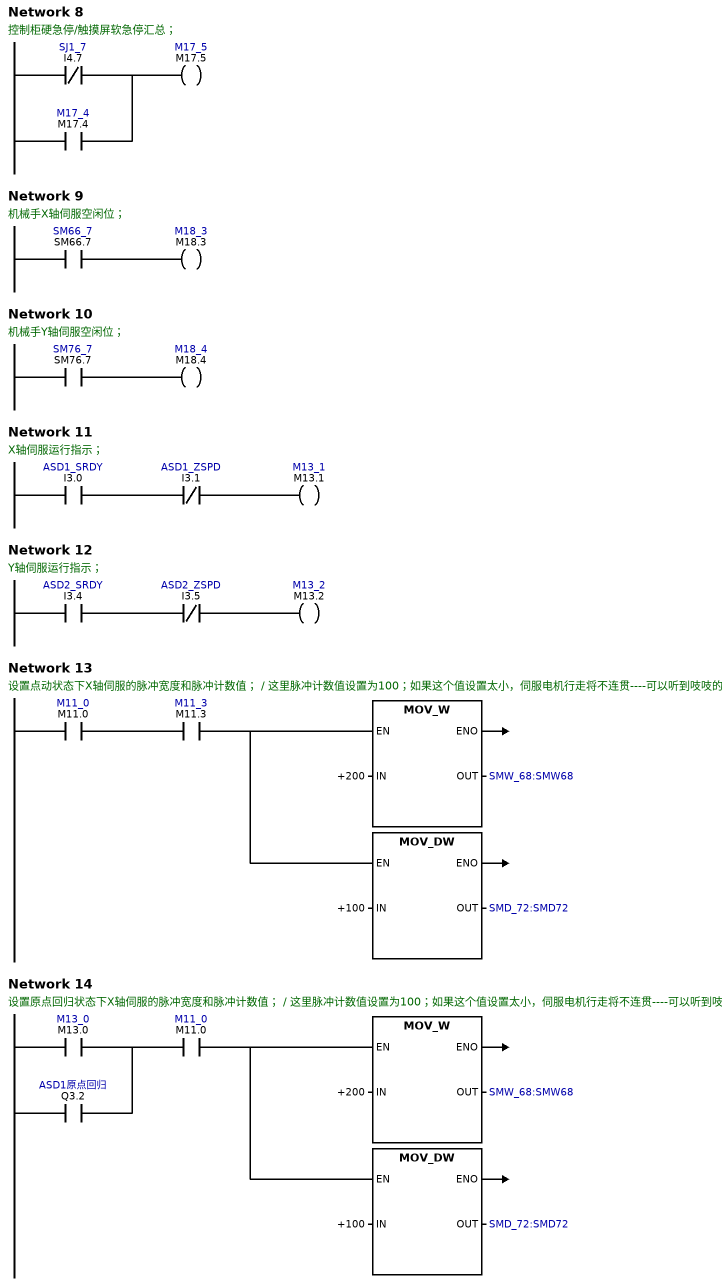
Network 8
// 控制柜硬急停/触摸屏软急停汇总；
LDN    SJ1_7:I4.7
O      M17_4:M17.4
=      M17_5:M17.5
Network 9
// 机械手X轴伺服空闲位；
LD     SM66_7:SM66.7
=      M18_3:M18.3
Network 10
// 机械手Y轴伺服空闲位；
LD     SM76_7:SM76.7
=      M18_4:M18.4
Network 11
// X轴伺服运行指示；
LD     ASD1_SRDY:I3.0
AN     ASD1_ZSPD:I3.1
=      M13_1:M13.1
Network 12
// Y轴伺服运行指示；
LD     ASD2_SRDY:I3.4
AN     ASD2_ZSPD:I3.5
=      M13_2:M13.2
Network 13
// 设置点动状态下X轴伺服的脉冲宽度和脉冲计数值；
// 这里脉冲计数值设置为100；如果这个值设置太小，伺服电机行走将不连贯----可以听到吱吱的刹车声。
// 点动时X轴伺服是缓慢运行的（脉冲周期为200微秒）；
LD     M11_0:M11.0
A      M11_3:M11.3
MOVW   +200, SMW_68:SMW68
MOVD   +100, SMD_72:SMD72
Network 14
// 设置原点回归状态下X轴伺服的脉冲宽度和脉冲计数值；
// 这里脉冲计数值设置为100；如果这个值设置太小，伺服电机行走将不连贯----可以听到吱吱的刹车声；
LD     M13_0:M13.0
O      ASD1原点回归:Q3.2
A      M11_0:M11.0
MOVW   +200, SMW_68:SMW68
MOVD   +100, SMD_72:SMD72
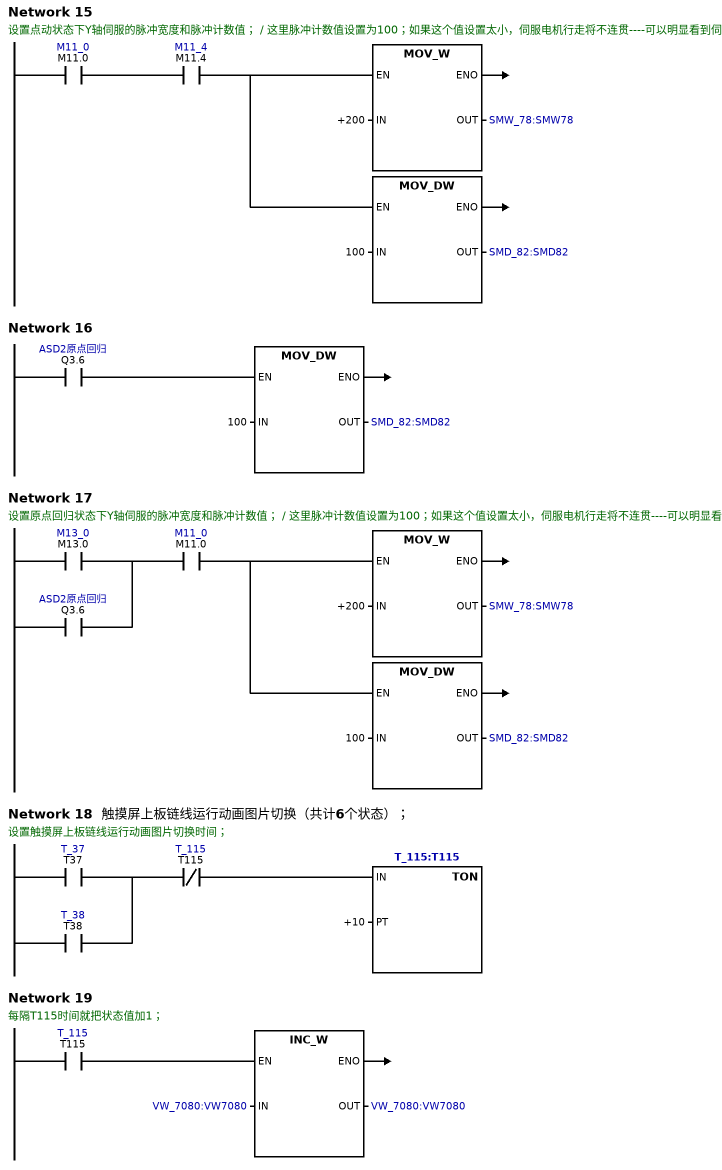
Network 15
// 设置点动状态下Y轴伺服的脉冲宽度和脉冲计数值；
// 这里脉冲计数值设置为100；如果这个值设置太小，伺服电机行走将不连贯----可以明显看到伺服停顿的现象；
// 点动时Y轴伺服是缓慢运行的（脉冲周期为150微秒）；
LD     M11_0:M11.0
A      M11_4:M11.4
MOVW   +200, SMW_78:SMW78
MOVD   100, SMD_82:SMD82
Network 16
LD     ASD2原点回归:Q3.6
MOVD   100, SMD_82:SMD82
Network 17
// 设置原点回归状态下Y轴伺服的脉冲宽度和脉冲计数值；
// 这里脉冲计数值设置为100；如果这个值设置太小，伺服电机行走将不连贯----可以明显看到伺服停顿的现象；
LD     M13_0:M13.0
O      ASD2原点回归:Q3.6
A      M11_0:M11.0
MOVW   +200, SMW_78:SMW78
MOVD   100, SMD_82:SMD82
Network 18 // 触摸屏上板链线运行动画图片切换（共计6个状态）；
// 设置触摸屏上板链线运行动画图片切换时间；
LD     T_37:T37
O      T_38:T38
AN     T_115:T115
TON    T_115:T115, +10
Network 19
// 每隔T115时间就把状态值加1；
LD     T_115:T115
INCW   VW_7080:VW7080
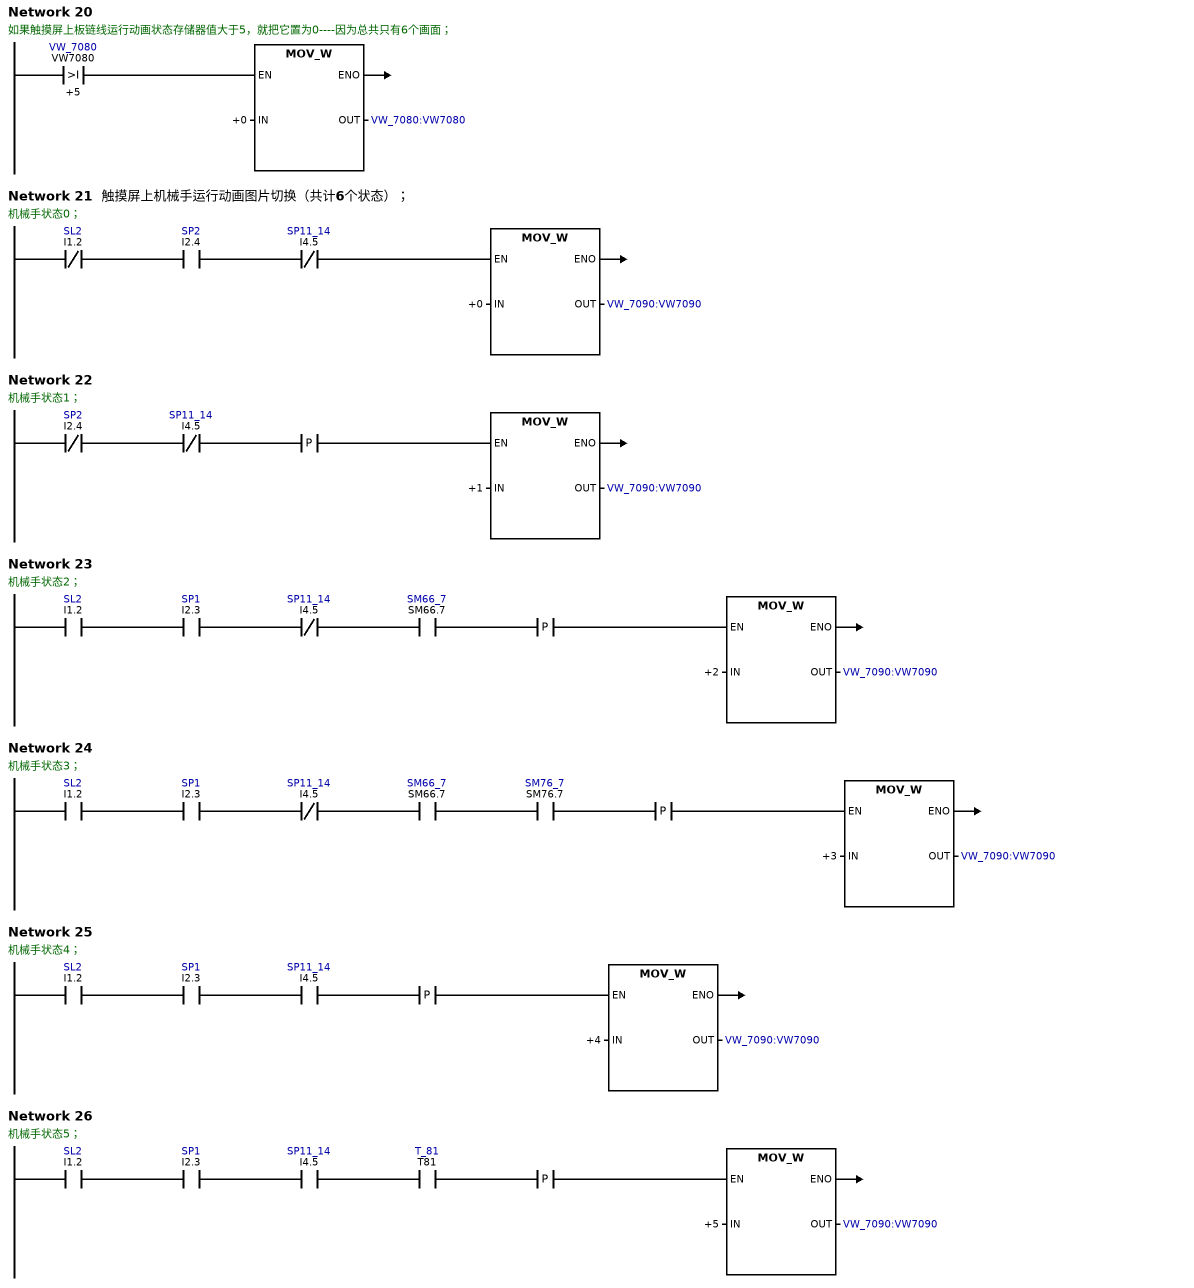
Network 20
// 如果触摸屏上板链线运行动画状态存储器值大于5，就把它置为0----因为总共只有6个画面；
LDW>   VW_7080:VW7080, +5
MOVW   +0, VW_7080:VW7080
Network 21 // 触摸屏上机械手运行动画图片切换（共计6个状态）；
// 机械手状态0；
LDN    SL2:I1.2
A      SP2:I2.4
AN     SP11_14:I4.5
MOVW   +0, VW_7090:VW7090
Network 22
// 机械手状态1；
LDN    SP2:I2.4
AN     SP11_14:I4.5
EU
MOVW   +1, VW_7090:VW7090
Network 23
// 机械手状态2；
LD     SL2:I1.2
A      SP1:I2.3
AN     SP11_14:I4.5
A      SM66_7:SM66.7
EU
MOVW   +2, VW_7090:VW7090
Network 24
// 机械手状态3；
LD     SL2:I1.2
A      SP1:I2.3
AN     SP11_14:I4.5
A      SM66_7:SM66.7
A      SM76_7:SM76.7
EU
MOVW   +3, VW_7090:VW7090
Network 25
// 机械手状态4；
LD     SL2:I1.2
A      SP1:I2.3
A      SP11_14:I4.5
EU
MOVW   +4, VW_7090:VW7090
Network 26
// 机械手状态5；
LD     SL2:I1.2
A      SP1:I2.3
A      SP11_14:I4.5
A      T_81:T81
EU
MOVW   +5, VW_7090:VW7090
END_SUBROUTINE_BLOCK

// SBR4: protected block, not included

// SBR5: protected block, not included

SUBROUTINE_BLOCK 机械手X轴伺服控制:SBR11
TITLE=S7-200控制台达伺服电机----机械手X轴伺服运动控制；
// 因为该工程要求的精度不高，所以直接采用晶体管输出型S7-200的Q0.0和Q0.1发送最高频率为20KHz的脉冲来控制伺服电机；如果输出频率不够，则在伺服驱动器中设置倍频来放大这个频率，不过这样的话控制精度也受到了影响（PLC发1个脉冲，伺服电机走了倍频值那么多步）；
// 该程序采用PTO脉冲串输出用于速度和位置控制；当然，PWM脉宽调制也可用于速度、位置或占空比控制，但其应用没有PTO方式那么广泛，因此该程序采用了PTO控制方式；
// 当组态一个输出为PTO操作时，生成一个50%占空比脉冲串用于步进电机或伺服电机的速度和位置的开环控制。内置PTO功能仅提供了脉冲串输出，您的应用程序必须通过PLC内置I/O或扩展模块提供方向和限位控制；
// 采用位置控制向导创建指令：只有勾选"使用高速计数器 HSC0（模式 12）自动计数线性 PTO 生成的脉冲。此功能将在内部完成，无需外部接线。"才会生成PTOx_LDPOS指令；        只有配置了运动包络，才会生成PTOx_RUN指令；        只有配置了"单速连续旋转"运动包络，而且勾选了"编一个子程序（PTOx_ADV）用于为此包络启动STOP（停止）操作。"才会生成PTOx_ADV子程序。
BEGIN
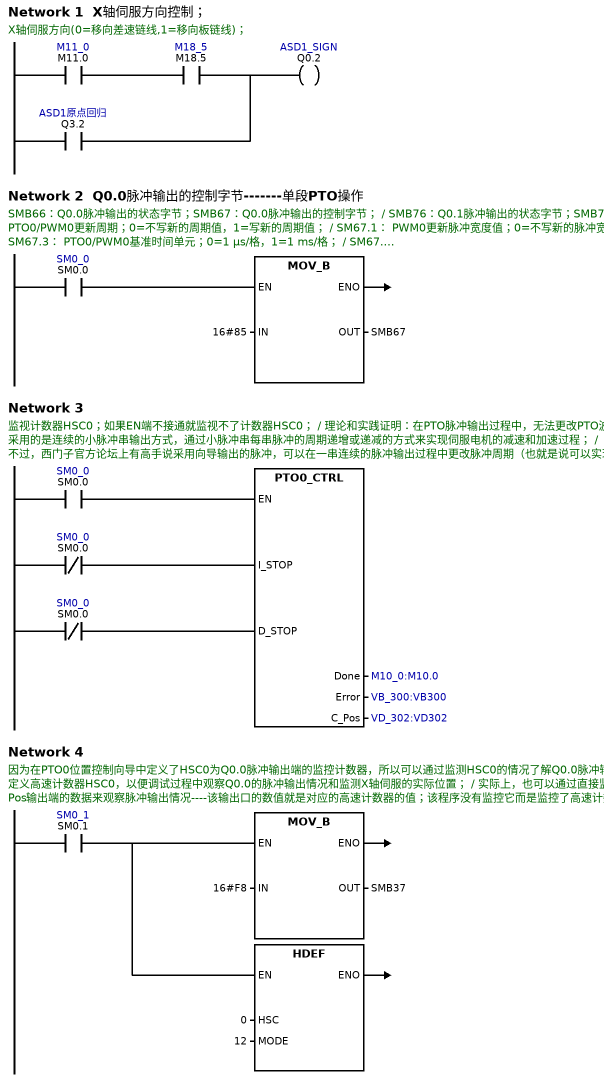
Network 1 // X轴伺服方向控制；
// X轴伺服方向(0=移向差速链线,1=移向板链线)；
LD     M11_0:M11.0
A      M18_5:M18.5
O      ASD1原点回归:Q3.2
=      ASD1_SIGN:Q0.2
Network 2 // Q0.0脉冲输出的控制字节-------单段PTO操作
// SMB66：Q0.0脉冲输出的状态字节；SMB67：Q0.0脉冲输出的控制字节；
// SMB76：Q0.1脉冲输出的状态字节；SMB77：Q0.1脉冲输出的控制字节；
// SM67.0： PTO0/PWM0更新周期；0=不写新的周期值，1=写新的周期值；
// SM67.1： PWM0更新脉冲宽度值；0=不写新的脉冲宽度，1=写新的脉冲宽度；
// SM67.2 ：PTO0更新脉冲量；0=不写新的脉冲量，1=写新的脉冲量；
// SM67.3： PTO0/PWM0基准时间单元；0=1 μs/格，1=1 ms/格；
// SM67.4 ：同步更新PWM0；0=异步更新，1=同步更新；当PLS指令执行时变化生效；如果改变了时间基准，会产生一个异步更新，而与PWM更新方式位的状态无关。有两个方法改变PWM波形的特性：
// 同步更新：如果不需要改变时间基准，就可以进行同步更新。利用同步更新，波形特性的变化发生在周期边沿，提供平滑转换。
//  异步更新：PWM的典型操作是当周期时间保持常数时变化脉冲宽度。所以，不需要改变时间基准。但是，如果需要改变PTO/PWM发生器的时间基准，就要使用异步更新。异步更新会造成PTO/PWM功能被瞬时禁止，和PWM波形不同步。这会引起被控设备的振动。由于这个原因，建议采用PWM同步更新。选择一个适合于所有周期时间的时间基准。
// SM67.5 ：PTO0操作：0=单段操作（周期和脉冲数存在SM存储器中），1=多段操作（包络表存在V存储器区）；
// SM67.6 ：PTO0/PWM0模式选择；0=PTO，1=PWM；
// SM67.7： PTO0/PWM0有效位；0=无效，1=有效；您可以在任意时刻禁止PTO或者PWM波形，方法为：首先将控制字节中的使能位（SM67.7或者SM77.7）清0，然后执行PLS指令；
// SMB67设置为2#10000101，即16#85；每次执行PLS前都写新的周期值和新的脉冲量，1 μs/格，单段操作（周期和脉冲数存在SM存储器中），PTO模式，PTO/PWM有效。
// PTO功能允许脉冲串“链接”或者“排队”。当当前脉冲串输出完成时，会立即开始输出一个新的脉冲串。这保证了多个输出脉冲串之间的连续性。
LD     SM0_0:SM0.0
MOVB   16#85, SMB67
Network 3
// 监视计数器HSC0；如果EN端不接通就监视不了计数器HSC0；
// 理论和实践证明：在PTO脉冲输出过程中，无法更改PTO波形的周期，也无法更改脉冲输出的个数；该程序没有采用向导的减速停止功能----采用的是连续的小脉冲串输出方式，通过小脉冲串每串脉冲的周期递增或递减的方式来实现伺服电机的减速和加速过程；
// 不过，西门子官方论坛上有高手说采用向导输出的脉冲，可以在一串连续的脉冲输出过程中更改脉冲周期（也就是说可以实现加速和减速过程）。不过笔者没有测试过，估计向导子程序采用的控制方式和笔者的小脉冲串输出方式原理上差不多。
LD     SM0_0:SM0.0
=      L60.0
LDN    SM0_0:SM0.0
=      L63.7
LDN    SM0_0:SM0.0
=      L63.6
LD     L60.0
CALL   PTO0_CTRL:SBR21, L63.7, L63.6, M10_0:M10.0, VB_300:VB300, VD_302:VD302
Network 4
// 因为在PTO0位置控制向导中定义了HSC0为Q0.0脉冲输出端的监控计数器，所以可以通过监测HSC0的情况了解Q0.0脉冲输出情况和监测X轴伺服的实际位置；
// 定义高速计数器HSC0，以便调试过程中观察Q0.0的脉冲输出情况和监测X轴伺服的实际位置；
// 实际上，也可以通过直接监视PTOX_CTRL的C Pos输出端的数据来观察脉冲输出情况----该输出口的数值就是对应的高速计数器的值；该程序没有监控它而是监控了高速计数器，只是采用了另外一种比较麻烦点的思路而已，不建议采用；
LD     SM0_1:SM0.1
MOVB   16#F8, SMB37
HDEF   0, 12
